	        #Retval := FC_LogMsg(EventID := 3002,
	                               EventLevel := 2,
	                               EventGroup := 33,
	                               LogMsg := DB_LogMsg.LogMsg_5);
	    END_IF;
	END_REGION
	
	//------------------------------------------------------
	// Log event when acknowledgment timeout occurs
	//------------------------------------------------------
	
	REGION Log event- acknowledgment timeout
	    IF #Communication.Log.Ack_timeout THEN
	        #Communication.Log.Ack_timeout := FALSE;
	        // Logging
	        //(LOG)3009=$ Node $, seq: $, acknowledge timeout!
	        DB_LogMsg.LogMsg_6.Para_STRING_01.Data := #Source.DecisionPoint;
	        DB_LogMsg.LogMsg_6.Para_BYTE_02.Data := #Communication.SendSeq;
	        #Retval := FC_LogMsg(EventID := 3009,
	                               EventLevel := 3,
	                               EventGroup := 33,
	                               LogMsg := DB_LogMsg.LogMsg_6);
	    END_IF;
	END_REGION
	
	
	
END_FUNCTION_BLOCK
END_NAMESPACE

NAMESPACE ProductionLine
FUNCTION_BLOCK FB_OPC_ReceiveSendAck
{ S7_Optimized_Access := 'TRUE' ; Published := 'FALSE' }
VERSION : 0.1
   VAR_IN_OUT 
      SourceSeq : Int;
      AckSeq : Int;
   END_VAR

   VAR 
      New_data_received : Bool;
      Ack_send : Bool;
      Log : Struct
         New_data_received : Bool;
         Ack_send : Bool;
      END_STRUCT;
   END_VAR


BEGIN
	// ==========================================================================================================================================
	// Company        : LogTech, s.r.o.
	// Created by     : Mahmoud Elnady
	// Block          : OPC_SendReciveAck
	// Project        : Lekarna, Chrudim -PLC001 -MCC001
	// Project number : 23-157
	// ==========================================================================================================================================
	
	// =========================
	// REGION: Acknowledgement Handling
	// =========================
	// This region handles sending an acknowledgment signal.
	// When #Ack_send is TRUE, it means an ACK needs to be sent for the last received sequence.
	// The ACK sequence is set equal to the source sequence to confirm receipt.
	// Then, #Ack_send is reset to FALSE, and a log flag is set to indicate ACK was sent.
	
	REGION Ack_Handling
	    
	    IF #Ack_send THEN
	        #AckSeq := #SourceSeq;        // Update ACK sequence to match source sequence
	        #Ack_send := FALSE;           // Reset ACK send request
	        #Log.Ack_send := TRUE;        // Set log flag for diagnostics or monitoring
	    END_IF;
	    
	END_REGION
	
	
	// =========================
	// REGION: New Data Detection
	// =========================
	// This region checks if a new data sequence has been received.
	// If the source and ACK sequences are not equal, it determines if it's truly new data:
	// - If both sequences are non-zero, or source is 1 and ACK is 0 (initial start case),
	//   then new data is considered received.
	// - Otherwise, it assumes the ACK was missed and sets ACK to current source.
	
	REGION New_Data_Detection
	    
	    IF #SourceSeq <> #AckSeq THEN
	        // Check if both sequences are valid (non-zero), or it's the initial case (1,0)
	        IF (#SourceSeq <> 0 AND #AckSeq <> 0) OR (#SourceSeq = 1 AND #AckSeq = 0) THEN
	            #New_data_received := TRUE;           // Flag new data received
	            #Log.#New_data_received := TRUE;      // Set log flag for diagnostics
	        ELSE
	            #AckSeq := #SourceSeq;                // Treat as missed ACK and sync
	        END_IF;
	    END_IF;
	    
	END_REGION
	
END_FUNCTION_BLOCK
END_NAMESPACE

NAMESPACE ProductionLine
FUNCTION_BLOCK FB_OPC_SendReciveAck
{ S7_Optimized_Access := 'TRUE' ; Published := 'FALSE' }
VERSION : 0.1
   VAR_INPUT 
      Timeout : Time;
   END_VAR

   VAR_IN_OUT 
      SourceSeq : Int;
      AckSeq : Int;
   END_VAR

   VAR 
      Send : Bool;
      New_Ack_received : Bool;
      Ack_timeout : Bool;
      Send_prev : Bool;
      SendSeq : Int;
      TimeoutTimmer {InstructionName := 'IEC_TIMER'; LibVersion := '1.0'; S7_SetPoint := 'False'} : IEC_TIMER;
      Log : Struct
         Send : Bool;
         New_Ack_received : Bool;
         Ack_timeout : Bool;
      END_STRUCT;
   END_VAR

   VAR CONSTANT 
      maxInc : Int := 9999;
   END_VAR


BEGIN
	// ==========================================================================================================================================
	// Company        : LogTech, s.r.o.
	// Created by     : Mahmoud Elnady
	// Block          : OPC_SendReciveAck
	// Project        : Lekarna, Chrudim -PLC001 -MCC001
	// Project number : 23-157
	// ==========================================================================================================================================
	
	// REGION: Handle New Send Request
	REGION Handle_Send_Request
	    // Triggered on rising edge of #Send signal
	    IF #Send AND NOT #Send_prev THEN
	         #AckSeq := 0;  // Reset acknowledgment sequence
	        
	        // Increment source sequence, wrapping around after 99999 (B#16#270F)
	         IF #SourceSeq <> #maxInc THEN
	             #SourceSeq += 1;
	         ELSE
	             #SourceSeq := 1;
	         END_IF;
	        
	        #SendSeq := #SourceSeq;       // Set current send sequence
	        #New_Ack_received := FALSE;   // Reset acknowledgment flag
	        #Log.Send := TRUE;            // Log send event
	    END_IF;
	END_REGION
	
	// REGION: Process Acknowledgment
	REGION Process_Acknowledgment
	    IF #Send THEN
	        // Check if acknowledgment is received for the current send
	        IF #AckSeq = #SendSeq THEN
	            IF #AckSeq <> 0 THEN
	                #New_Ack_received := TRUE;     // Mark new acknowledgment
	                #Ack_timeout := FALSE;         // Clear timeout flag
	                #Log.#New_Ack_received := TRUE; // Log acknowledgment
	            END_IF;
	            //#Send := FALSE;  // Reset send signal
	        END_IF;
	    END_IF;
	    
	    // Update previous send state
	    #Send_prev := #Send;
	END_REGION
	
	
	// REGION: Timeout Management and Retransmission
	REGION Handle_Send_Timeout
	    // Activate timeout timer if timeout value is set
	    IF #Timeout <> T#0s THEN
	        #TimeoutTimmer.TON(IN := #Send AND NOT #New_Ack_received ,
	                           PT := #Timeout);
	    END_IF;
	    
	    // On timeout expiration, trigger retransmission logic
	    IF #TimeoutTimmer.Q THEN
	        #Send_prev := FALSE;         // Reset previous send to retrigger
	        #Ack_timeout := TRUE;        // Mark acknowledgment timeout
	        #Log.Ack_timeout := TRUE;    // Log timeout event
	        RESET_TIMER(#TimeoutTimmer); // Reset timer
	    END_IF;
	END_REGION
	
	
	
	
END_FUNCTION_BLOCK
END_NAMESPACE

NAMESPACE ProductionLine
FUNCTION_BLOCK FB_OPC_SysStatus
{ S7_Optimized_Access := 'TRUE' ; Published := 'FALSE' }
VERSION : 0.1
   VAR_IN_OUT 
      Source : OPC_SystemStatus;
      Ack : OPC_SystStatus_Ack;
   END_VAR

   VAR 
      Comm { S7_SetPoint := 'False'} : FB_OPC_SendReciveAck;
      staSource { ExternalAccessible := 'False'; ExternalVisible := 'False'; ExternalWritable := 'False'; S7_SetPoint := 'False'} : OPC_SystemStatus;
      staAck { ExternalAccessible := 'False'; ExternalVisible := 'False'; ExternalWritable := 'False'; S7_SetPoint := 'False'} : OPC_SystStatus_Ack;
   END_VAR

   VAR_TEMP 
      Retval : Int;
   END_VAR


BEGIN
	// ==========================================================================================================================================
	// Company        : LogTech, s.r.o.
	// Created by     : Mahmoud Elnady
	// Block          : OPC_SendReciveAck
	// Project        : Lekarna, Chrudim -PLC001 -MCC001
	// Project number : 23-157
	// ==========================================================================================================================================
	
	//======================================================
	// Region: Communication Handling and Logging
	// Description: Manages the communication routine and logs
	//              events for message sending, acknowledgment
	//              reception, and acknowledgment timeout.
	//======================================================
	   
	//------------------------------------------------------
	// Call communication routine
	//------------------------------------------------------
	REGION Communication Routine
	    #Comm(SourceSeq := #staSource.SourceSeq,
	          AckSeq := #staAck.AckSeq,
	             Timeout := T#20s);
	END_REGION
	
	#Source.SourceSeq := #staSource.SourceSeq;
	#staAck.AckSeq := #Ack.AckSeq;
	
	
	//------------------------------------------------------
	// Log event when a new message is sent
	//------------------------------------------------------
	REGION Log event - new message
	    IF #Comm.Log.Send THEN
	        #Comm.Log.Send := FALSE;
	        
	        // (LOG)3001=$ Node $, new message sent, seq: $, $ $ $ $ $ $ $ $, $ $ $ $ $ $ $ $ $ $ $ $ $ $ $ $
	        DB_LogMsg.LogMsg_1.Para_BYTE_02.Data := #Source.SourceSeq;
	        
	        // Call logging function
	        #Retval := FC_LogMsg(EventID := 3007,
	                               EventLevel := 2,
	                               EventGroup := 33,
	                               LogMsg := DB_LogMsg.LogMsg_1);
	    END_IF;
	END_REGION
	
	   
	//------------------------------------------------------
	// Log event when new acknowledgment is received
	//------------------------------------------------------
	REGION  Log event-New acknowledgment
	       IF #Comm.Log.New_Ack_received THEN
	           #Comm.Log.New_Ack_received := FALSE;
	           
	           // (LOG)3008=$ Node $, acknowledge received, seq: $, WMSID: $
	           DB_LogMsg.LogMsg_2.Para_BYTE_02.Data := #Ack.AckSeq;
	           
	           // Call logging function
	           #Retval := FC_LogMsg(EventID := 3008,
	                                  EventLevel := 2,
	                                  EventGroup := 33,
	                                  LogMsg := DB_LogMsg.LogMsg_2);
	       END_IF;
	END_REGION
	
	   
	//------------------------------------------------------
	// Log event when acknowledgment timeout occurs
	//------------------------------------------------------
	REGION Log event- acknowledgment timeout
	       IF #Comm.Log.Ack_timeout THEN
	           #Comm.Log.Ack_timeout := FALSE;
	           
	           // (LOG)3009=$ Node $, seq: $, acknowledge timeout!
	           DB_LogMsg.LogMsg_3.Para_BYTE_02.Data := #Comm.SendSeq;
	           
	           // Call logging function
	           #Retval := FC_LogMsg(EventID := 3009,
	                                  EventLevel := 3,
	                                  EventGroup := 33,
	                                  LogMsg := DB_LogMsg.LogMsg_3);
	       END_IF;
	END_REGION
	    
	
	   
	   
	
END_FUNCTION_BLOCK
END_NAMESPACE

NAMESPACE ProductionLine
FUNCTION_BLOCK FB_Segments
{ S7_Optimized_Access := 'TRUE' ; Published := 'FALSE' }
VERSION : 0.1
   VAR 
      ConveyorID : Int;
      "Counter" : Int;
      FlowRackLoop1 : Array[_."B1.1.1".._."B1.23.1"] of Bool;
      FlowRackLoop2 : Array[_."B1.6.1".._."B1.18.1"] of Bool;
      Fragileloop1 : Array[_."D1.1.1".._."E1.6.1"] of Bool;
      Fragileloop2 : Array[_."D1.9.1".._."D1.10.1"] of Bool;
      cmp : Struct
         FlowRackLoop1 : Array[_."B1.1.1".._."B1.23.1"] of Bool;
         FlowRackLoop2 : Array[_."B1.6.1".._."B1.18.1"] of Bool;
         Fragileloop1 : Array[_."D1.1.1".._."E1.6.1"] of Bool;
         Fragileloop2 : Array[_."D1.9.1".._."D1.10.1"] of Bool;
      END_STRUCT;
      FlowRackLoopReadyToRun : Bool;
      FlowRackWorkPlaceLeftReadyToRun : Bool;
      FlowRackWorkPlaceRightReadyToRun : Bool;
      FragileloopReadyToRun : Bool;
   END_VAR


BEGIN
	// ==========================================================================================================================================
	// Company        : LogTech, s.r.o.
	// Created by     : Mahmoud Elnady
	// Block          : FB_Segments
	// Project        : Lekarna, Chrudim -PLC001 -MCC001
	// Project number : 23-157
	// ==========================================================================================================================================
	
	// ===============================
	// REGION: Flow rack loop
	// Purpose: Check the ReadyToRun status of conveyors and transfer units 
	//          for a flow rack section, then compare with a stored snapshot.
	// ===============================
	REGION Flow rack loop
	    
	    // ---------------------------------
	    // REGION: Conveyor Status Loop
	    // Purpose: Iterate over conveyor IDs from B1.1.1 to B1.28.1 
	    //          and store their ReadyToRun status in FlowRackLoop1 array.
	    // ---------------------------------
	   REGION Conveyor Status
	        FOR #Counter := _."B1.1.1" TO _."B1.23.1" DO
	            // Store ReadyToRun status of the current conveyor into FlowRackLoop1
	            #FlowRackLoop1[#Counter] := 
	            _.Global.DB_Global.Status.Line.ProductionLine.ReadyToRun[#Counter];
	        END_FOR;
	    END_REGION
	   
	    // ---------------------------------
	    // REGION: Transfer Unit Status Loop
	    // Purpose: Iterate over transfer unit IDs from B1.6.1 to B1.21.1 
	    //          and store their ReadyToRun status in FlowRackLoop2 array.
	    // ---------------------------------
	    REGION TransferUnit Status
	        FOR #Counter := _."B1.6.1" TO _."B1.18.1" DO
	            // Store ReadyToRun status of the current transfer unit into FlowRackLoop2
	            #FlowRackLoop2[#Counter] :=
	            _.Global.DB_Global.Status.Line.ProductionLine.ReadyToRun[#Counter];
	        END_FOR;
	    END_REGION
	    
	    // ---------------------------------
	    // REGION: Status Comparison
	    // Purpose: Check if both conveyor and transfer unit statuses 
	    //          match the previous recorded values (#cmp arrays).
	    // ---------------------------------
	    REGION Comparison
	        #FlowRackLoopReadyToRun := NOT 
	        ((#cmp.FlowRackLoop1 = #FlowRackLoop1) AND
	        (#cmp.FlowRackLoop2 = #FlowRackLoop2));
	    END_REGION
	    
	END_REGION
	
	
	// ===============================
	// REGION: Flow rack work place left
	// Purpose: ReadyToRun check for two specific conveyors on the left side.
	// ===============================
	REGION Flow rack work place left
	    #FlowRackWorkPlaceLeftReadyToRun :=
	    _.Global.DB_Global.Status.Line.ProductionLine.ReadyToRun[_."C1.4.1"] AND
	    _.Global.DB_Global.Status.Line.ProductionLine.ReadyToRun[_."C1.4.2"];
	END_REGION
	
	
	// ===============================
	// REGION: Flow rack work place right
	// Purpose: ReadyToRun check for two specific conveyors on the right side.
	// ===============================
	REGION Flow rack work place right
	    #FlowRackWorkPlaceRightReadyToRun :=
	    _.Global.DB_Global.Status.Line.ProductionLine.ReadyToRun[_."C1.2.1"] AND
	    _.Global.DB_Global.Status.Line.ProductionLine.ReadyToRun[_."C1.2.2"];
	END_REGION
	
	
	// ===============================
	// REGION: Fragile loop
	// Purpose: Same logic as Flow rack loop, but for the "fragile" product path.
	// ===============================
	REGION Fragile loop
	    
	    // ---------------------------------
	    // REGION: Conveyor Status Loop (Fragile)
	    // Purpose: Store ReadyToRun status for conveyors D1.1.1 to E1.6.1
	    // ---------------------------------
	    REGION Conveyor Status
	        FOR #Counter := _."D1.1.1" TO _."E1.6.1" DO
	            #Fragileloop1[#Counter] :=
	            _.Global.DB_Global.Status.Line.ProductionLine.ReadyToRun[#Counter];
	        END_FOR;
	    END_REGION
	    
	    // ---------------------------------
	    // REGION: Transfer Unit Status Loop (Fragile)
	    // Purpose: Store ReadyToRun status for transfer units D1.8.1 to D1.9.1
	    // ---------------------------------
	    REGION TransferUnit Status
	        FOR #Counter := _."D1.9.1" TO _."D1.10.1" DO
	            #Fragileloop2[#Counter] :=
	            _.Global.DB_Global.Status.Line.ProductionLine.ReadyToRun[#Counter];
	        END_FOR;
	    END_REGION
	    
	    // ---------------------------------
	    // REGION: Status Comparison (Fragile)
	    // Purpose: Check if current fragile loop status matches previous snapshot.
	    // ---------------------------------
	    REGION Comparison
	        #FragileloopReadyToRun := NOT
	        ((#cmp.Fragileloop1 = #Fragileloop1) AND
	        (#cmp.Fragileloop2 = #Fragileloop2));
	    END_REGION
	    
	END_REGION
	
END_FUNCTION_BLOCK
END_NAMESPACE

NAMESPACE ProductionLine
FUNCTION_BLOCK FB_Technology
{ S7_Optimized_Access := 'TRUE' ; Published := 'FALSE' }
VERSION : 0.1
   VAR 
      IP11 : String := 'IP11';
      IP12 : String := 'IP12';
      IP21 : String := 'IP21';
      IP22 : String := 'IP22';
      IP23 : String := 'IP23';
      IP31 : String := 'IP31';
      IP32 : String := 'IP32';
      IP41 : String := 'IP41';
      IP42 : String := 'IP42';
      ComDownStream : Struct
         DP1 : Bool;
         DP2 : Bool;
         DP3 : Bool;
         DP4 : Bool;
      END_STRUCT;
      ComTimmerDP1 {InstructionName := 'TON_TIME'; LibVersion := '1.0'} : TON_TIME;
      ComTimmerDP2 {InstructionName := 'TON_TIME'; LibVersion := '1.0'} : TON_TIME;
      ComTimmerDP3 {InstructionName := 'TON_TIME'; LibVersion := '1.0'} : TON_TIME;
      ComTimmerDP4 {InstructionName := 'TON_TIME'; LibVersion := '1.0'} : TON_TIME;
   END_VAR


BEGIN
	// ==========================================================================================================================================
	// Company        : LogTech, s.r.o.
	// Created by     : Mahmoud Elnady
	// Block          : FB_OPC_Communication
	// Project        : Lekarna, Chrudim -PLC001 -MCC001
	// Project number : 23-157
	// ==========================================================================================================================================
	
	REGION Destination request TO WMS
	    // Send destination request to WMS
	    REGION DP1
	        IF IDB_BarcodeReader.DP1."Dataman-Results Available" OR
	            IDB_ProductionLine."A1.5.1".CONVEYOR_SENSOR.PosEdge.Q
	        THEN
	            OPC_Data.DP1.DestRequest.Source.Barcode := IDB_BarcodeReader.DP1.ResultStr;
	            IDB_OPC_Communication.Communication_DP1.Communication.Send := TRUE;
	            #ComDownStream.DP1 := TRUE;
	        ELSIF (IDB_OPC_Communication.Communication_DP1.Communication.SourceSeq =
	            IDB_OPC_Communication.Communication_DP1.Communication.AckSeq)
	            OR #ComTimmerDP1.Q
	        THEN
	            IDB_OPC_Communication.Communication_DP1.Communication.Send := FALSE;
	        END_IF;
	         
	    END_REGION
	    
	    REGION DP2
	        IF IDB_BarcodeReader.DP2."Dataman-Results Available" OR
	            IDB_ProductionLine."B1.9.1".CONVEYOR_SENSOR.PosEdge.Q
	        THEN
	            OPC_Data.DP2.DestRequest.Source.Barcode := IDB_BarcodeReader.DP2.ResultStr;
	            IDB_OPC_Communication.Communication_DP2.Communication.Send := TRUE;
	            #ComDownStream.DP2 := TRUE;
	        ELSIF (IDB_OPC_Communication.Communication_DP2.Communication.SourceSeq =
	            IDB_OPC_Communication.Communication_DP2.Communication.AckSeq)
	            OR #ComTimmerDP2.Q
	        THEN
	            IDB_OPC_Communication.Communication_DP2.Communication.Send := FALSE;
	        END_IF;
	    END_REGION
	    
	    REGION DP3
	        IF IDB_BarcodeReader.DP3."Dataman-Results Available" OR
	            IDB_ProductionLine."B1.17.1".CONVEYOR_SENSOR.PosEdge.Q
	        THEN
	            OPC_Data.DP3.DestRequest.Source.Barcode := IDB_BarcodeReader.DP3.ResultStr;
	            IDB_OPC_Communication.Communication_DP3.Communication.Send := TRUE;
	            #ComDownStream.DP3 := TRUE;
	        ELSIF (IDB_OPC_Communication.Communication_DP3.Communication.SourceSeq =
	            IDB_OPC_Communication.Communication_DP3.Communication.AckSeq)
	            OR #ComTimmerDP3.Q
	        THEN
	            IDB_OPC_Communication.Communication_DP3.Communication.Send := FALSE;
	        END_IF;
	    END_REGION
	    
	    REGION DP4
	        IF IDB_BarcodeReader.DP4."Dataman-Results Available" OR
	            IDB_ProductionLine."A1.7.4".CONVEYOR_SENSOR.PosEdge.Q
	        THEN
	            OPC_Data.DP4.DestRequest.Source.Barcode := IDB_BarcodeReader.DP4.ResultStr;
	            IDB_OPC_Communication.Communication_DP4.Communication.Send := TRUE;
	            #ComDownStream.DP4 := TRUE;
	        ELSIF (IDB_OPC_Communication.Communication_DP4.Communication.SourceSeq =
	            IDB_OPC_Communication.Communication_DP4.Communication.AckSeq)
	            OR #ComTimmerDP4.Q
	        THEN
	            IDB_OPC_Communication.Communication_DP4.Communication.Send := FALSE;
	        END_IF;
	        
	    END_REGION
	    
	END_REGION
	
	REGION Wait FOR data from WMS
	    // Wait for data from WMS
	    REGION Mabs A1.6.1 & A1.6.2 Dir
	        IF IDB_OPC_Communication.Communication_DP1.Communication.New_Ack_received THEN
	            //IDB_OPC_Communication.Communication_DP1.Communication.New_Ack_received := FALSE;
	            #ComDownStream.DP1 := FALSE;
	            IF OPC_Data.DP1.DestRequest.Ack.Destination = #IP11 THEN
	                DB_ToteTracking.Conveyor[_."A1.5.1"].ToteDir.Straight := TRUE;
	                DB_ToteTracking.Conveyor[_."A1.5.1"].ToteDir.toRight := FALSE;
	                DB_ToteTracking.Conveyor[_."A1.2.1"].ToteDir.toLeft := FALSE;
	            ELSIF
	                OPC_Data.DP1.DestRequest.Ack.Destination = #IP12 THEN
	                DB_ToteTracking.Conveyor[_."A1.5.1"].ToteDir.toRight := TRUE;
	                DB_ToteTracking.Conveyor[_."A1.5.1"].ToteDir.Straight := FALSE;
	                DB_ToteTracking.Conveyor[_."A1.5.1"].ToteDir.toLeft := FALSE;
	            ELSE
	                DB_ToteTracking.Conveyor[_."A1.5.1"].ToteDir.Straight := FALSE;
	                DB_ToteTracking.Conveyor[_."A1.5.1"].ToteDir.toRight := FALSE;
	                DB_ToteTracking.Conveyor[_."A1.5.1"].ToteDir.toLeft := FALSE;
	            END_IF;
	        END_IF;
	    END_REGION
	    
	    REGION Transfer Unit B1.10.1 Dir
	        IF IDB_OPC_Communication.Communication_DP2.Communication.New_Ack_received THEN
	            //IDB_OPC_Communication.Communication_DP2.Communication.New_Ack_received := FALSE;
	            #ComDownStream.DP2 := FALSE;
	            IF  OPC_Data.DP2.DestRequest.Ack.Destination = #IP21 THEN
	                DB_ToteTracking.Conveyor[_."B1.9.1"].ToteDir.Straight := TRUE;
	                DB_ToteTracking.Conveyor[_."B1.9.1"].ToteDir.toRight := FALSE;
	                DB_ToteTracking.Conveyor[_."B1.9.1"].ToteDir.toLeft := FALSE;
	            ELSIF
	                (OPC_Data.DP2.DestRequest.Ack.Destination = #IP22 OR
	                OPC_Data.DP2.DestRequest.Ack.Destination = #IP23) THEN
	                DB_ToteTracking.Conveyor[_."B1.9.1"].ToteDir.toRight := TRUE;
	                DB_ToteTracking.Conveyor[_."B1.9.1"].ToteDir.Straight := FALSE;
	                DB_ToteTracking.Conveyor[_."B1.9.1"].ToteDir.toLeft := FALSE;
	                //Transfer Unit C1.1.3 Dir
	                IF OPC_Data.DP2.DestRequest.Ack.Destination = #IP22 THEN
	                    DB_ToteTracking.Transfer[_."B1.9.1"].Straight := FALSE;
	                    DB_ToteTracking.Transfer[_."B1.9.1"].toRight := TRUE;
	                    DB_ToteTracking.Transfer[_."B1.9.1"].toLeft := FALSE;
	                ELSIF  OPC_Data.DP2.DestRequest.Ack.Destination = #IP23 THEN
	                    DB_ToteTracking.Transfer[_."B1.9.1"].toRight := FALSE;
	                    DB_ToteTracking.Transfer[_."B1.9.1"].Straight := FALSE;
	                    DB_ToteTracking.Transfer[_."B1.9.1"].toLeft := TRUE;
	                ELSE
	                    DB_ToteTracking.Transfer[_."B1.9.1"].Straight := FALSE;
	                    DB_ToteTracking.Transfer[_."B1.9.1"].toRight := FALSE;
	                    DB_ToteTracking.Transfer[_."B1.9.1"].toLeft := FALSE;
	                END_IF;
	                
	            ELSE
	                DB_ToteTracking.Conveyor[_."B1.9.1"].ToteDir.Straight := FALSE;
	                DB_ToteTracking.Conveyor[_."B1.9.1"].ToteDir.toRight := FALSE;
	                DB_ToteTracking.Conveyor[_."B1.9.1"].ToteDir.toLeft := FALSE;
	            END_IF;
	        END_IF;
	    END_REGION
	    
	    
	    REGION Transfer Unit B1.21.1 Dir
	        IF IDB_OPC_Communication.Communication_DP3.Communication.New_Ack_received THEN
	            //IDB_OPC_Communication.Communication_DP3.Communication.New_Ack_received := FALSE;
	            #ComDownStream.DP3 := FALSE;
	            IF  OPC_Data.DP3.DestRequest.Ack.Destination = #IP31 THEN
	                DB_ToteTracking.Conveyor[_."B1.17.1"].ToteDir.Straight := TRUE;
	                DB_ToteTracking.Conveyor[_."B1.17.1"].ToteDir.toRight := FALSE;
	                DB_ToteTracking.Conveyor[_."B1.17.1"].ToteDir.toLeft := FALSE;
	                
	            ELSIF OPC_Data.DP3.DestRequest.Ack.Destination = #IP32 THEN
	                DB_ToteTracking.Conveyor[_."B1.17.1"].ToteDir.toRight := FALSE;
	                DB_ToteTracking.Conveyor[_."B1.17.1"].ToteDir.Straight := FALSE;
	                DB_ToteTracking.Conveyor[_."B1.17.1"].ToteDir.toLeft := TRUE;
	                
	            ELSE
	                DB_ToteTracking.Conveyor[_."B1.17.1"].ToteDir.Straight := FALSE;
	                DB_ToteTracking.Conveyor[_."B1.17.1"].ToteDir.toRight := FALSE;
	                DB_ToteTracking.Conveyor[_."B1.17.1"].ToteDir.toLeft := FALSE;
	            END_IF;
	        END_IF;
	    END_REGION
	    
	    REGION Mabs A1.8.1 & A1.8.2 Dir
	        IF IDB_OPC_Communication.Communication_DP4.Communication.New_Ack_received THEN
	            //IDB_OPC_Communication.Communication_DP4.Communication.New_Ack_received := FALSE;
	            #ComDownStream.DP4 := FALSE;
	            IF  OPC_Data.DP4.DestRequest.Ack.Destination = #IP41 THEN
	                DB_ToteTracking.Conveyor[_."A1.7.4"].ToteDir.Straight := TRUE;
	                DB_ToteTracking.Conveyor[_."A1.7.4"].ToteDir.toRight := FALSE;
	                DB_ToteTracking.Conveyor[_."A1.7.4"].ToteDir.toLeft := FALSE;
	            ELSIF
	                OPC_Data.DP4.DestRequest.Ack.Destination = #IP42 THEN
	                DB_ToteTracking.Conveyor[_."A1.7.4"].ToteDir.toRight := TRUE;
	                DB_ToteTracking.Conveyor[_."A1.7.4"].ToteDir.Straight := FALSE;
	                DB_ToteTracking.Conveyor[_."A1.7.4"].ToteDir.toLeft := FALSE;
	            ELSE
	                DB_ToteTracking.Conveyor[_."A1.7.4"].ToteDir.Straight := FALSE;
	                DB_ToteTracking.Conveyor[_."A1.7.4"].ToteDir.toRight := FALSE;
	                DB_ToteTracking.Conveyor[_."A1.7.4"].ToteDir.toLeft := FALSE;
	            END_IF;
	        END_IF;
	    END_REGION
	    
	    REGION Wait WMS Response
	        #ComTimmerDP1(IN := #ComDownStream.DP1,
	                      PT := t#45s);
	        
	        IF #ComTimmerDP1.Q THEN
	            #ComDownStream.DP1 := FALSE;
	        END_IF;
	        
	        #ComTimmerDP2(IN := #ComDownStream.DP2,
	                      PT := t#45s);
	        
	        IF #ComTimmerDP2.Q THEN
	            #ComDownStream.DP2 := FALSE;
	        END_IF;
	        
	        #ComTimmerDP3(IN := #ComDownStream.DP3,
	                      PT := t#45s);
	        
	        IF #ComTimmerDP3.Q THEN
	            #ComDownStream.DP3 := FALSE;
	        END_IF;
	        
	        #ComTimmerDP4(IN := #ComDownStream.DP4,
	                      PT := t#45s);
	        
	        IF #ComTimmerDP4.Q THEN
	            #ComDownStream.DP4 := FALSE;
	        END_IF;
	        
	    END_REGION
	
	END_REGION
	
	
	REGION Destination info TO WMS
	    // Send destination info to WMS
	    REGION IP1
	        IF IDB_ProductionLine."A1.7.2".CONVEYOR_SENSOR.PosEdge.Q AND
	            NOT IDB_OPC_Communication.Communication_IP1.Communication.Send THEN
	            OPC_Data.IP1.DestInfo.Source.Barcode := DB_ToteTracking.Conveyor[_."A1.7.1"].Barcode;
	            OPC_Data.IP1.DestInfo.Source.InformationPoint := #IP11;
	            IDB_OPC_Communication.Communication_IP1.Communication.Send := TRUE;
	        END_IF;
	        
	    END_REGION
	    REGION IP2
	        IF IDB_ProductionLine."B1.2.1".CONVEYOR_SENSOR.PosEdge.Q AND
	            NOT IDB_OPC_Communication.Communication_IP2.Communication.Send THEN
	            OPC_Data.IP2.DestInfo.Source.Barcode := DB_ToteTracking.Conveyor[_."B1.1.1"].Barcode;
	            OPC_Data.IP2.DestInfo.Source.InformationPoint := #IP12;
	            IDB_OPC_Communication.Communication_IP2.Communication.Send := TRUE;
	        END_IF;
	        
	    END_REGION
	    
	    REGION IP3
	        IF IDB_ProductionLine."B1.11.2".CONVEYOR_SENSOR.PosEdge.Q AND
	            NOT IDB_OPC_Communication.Communication_IP3.Communication.Send THEN
	            OPC_Data.IP3.DestInfo.Source.Barcode := DB_ToteTracking.Conveyor[_."B1.11.1"].Barcode;
	            OPC_Data.IP3.DestInfo.Source.InformationPoint := #IP21;
	            IDB_OPC_Communication.Communication_IP3.Communication.Send := TRUE;
	        END_IF;
	    END_REGION
	    
	    REGION IP4
	        IF IDB_ProductionLine."C1.2.1".CONVEYOR_SENSOR.PosEdge.Q AND
	            NOT IDB_OPC_Communication.Communication_IP4.Communication.Send THEN
	            OPC_Data.IP4.DestInfo.Source.Barcode := DB_ToteTracking.Conveyor[_."C1.2.2"].Barcode;
	            OPC_Data.IP4.DestInfo.Source.InformationPoint := #IP22;
	            IDB_OPC_Communication.Communication_IP4.Communication.Send := TRUE;
	        END_IF;
	        
	    END_REGION
	    
	    REGION IP5
	        IF IDB_ProductionLine."C1.4.2".CONVEYOR_SENSOR.PosEdge.Q AND
	            NOT IDB_OPC_Communication.Communication_IP5.Communication.Send THEN
	            OPC_Data.IP5.DestInfo.Source.Barcode := DB_ToteTracking.Conveyor[_."C1.4.1"].Barcode;
	            OPC_Data.IP5.DestInfo.Source.InformationPoint := #IP23;
	            IDB_OPC_Communication.Communication_IP5.Communication.Send := TRUE;
	        END_IF;
	        
	    END_REGION
	    
	    REGION IP6
	        IF IDB_ProductionLine."B1.20.1".CONVEYOR_SENSOR.PosEdge.Q AND
	            NOT IDB_OPC_Communication.Communication_IP6.Communication.Send THEN
	            OPC_Data.IP6.DestInfo.Source.Barcode := DB_ToteTracking.Conveyor[_."B1.19.1"].Barcode;
	            OPC_Data.IP6.DestInfo.Source.InformationPoint := #IP31;
	            IDB_OPC_Communication.Communication_IP6.Communication.Send := TRUE;
	        END_IF;
	    END_REGION
	    
	    REGION IP7
	        IF (IDB_ProductionLine."B1.6.1"."Left/RightSensor" OR 
	            _.ProductionLine.IDB_Flow_Test.R_TRIG_Instance.Q) AND //only for simulation purpose 
	            NOT IDB_OPC_Communication.Communication_IP7.Communication.Send THEN
	            OPC_Data.IP7.DestInfo.Source.Barcode := DB_ToteTracking.Conveyor[_."B1.6.1"].Barcode;
	            OPC_Data.IP7.DestInfo.Source.InformationPoint := #IP32;
	            IDB_OPC_Communication.Communication_IP7.Communication.Send := TRUE;
	        END_IF;
	        
	    END_REGION
	    
	    REGION IP8
	        IF IDB_ProductionLine."A1.10.2".CONVEYOR_SENSOR.PosEdge.Q AND
	            NOT IDB_OPC_Communication.Communication_IP8.Communication.Send THEN
	            OPC_Data.IP8.DestInfo.Source.Barcode := DB_ToteTracking.Conveyor[_."A1.10.1"].Barcode;
	            OPC_Data.IP8.DestInfo.Source.InformationPoint := #IP41;
	            IDB_OPC_Communication.Communication_IP8.Communication.Send := TRUE;
	        END_IF;
	    END_REGION
	    
	    REGION IP9
	        IF IDB_ProductionLine."D1.2.1".CONVEYOR_SENSOR.PosEdge.Q AND
	            NOT IDB_OPC_Communication.Communication_IP9.Communication.Send THEN
	            OPC_Data.IP9.DestInfo.Source.Barcode := DB_ToteTracking.Conveyor[_."D1.1.1"].Barcode;
	            OPC_Data.IP9.DestInfo.Source.InformationPoint := #IP42;
	            IDB_OPC_Communication.Communication_IP9.Communication.Send := TRUE;
	        END_IF;
	    END_REGION
	    
	    
	END_REGION
	
	
	REGION Wait FOR data from WMS
	    // Wait for data from WMS
	    REGION IP1 Ack
	        IF IDB_OPC_Communication.Communication_IP1.Communication.New_Ack_received THEN
	            IDB_OPC_Communication.Communication_IP1.Communication.Send := FALSE;
	            IDB_OPC_Communication.Communication_IP1.Communication.New_Ack_received := FALSE;
	        END_IF;
	    END_REGION
	    
	    REGION IP2 Ack
	        IF IDB_OPC_Communication.Communication_IP2.Communication.New_Ack_received THEN
	            IDB_OPC_Communication.Communication_IP2.Communication.Send := FALSE;
	            IDB_OPC_Communication.Communication_IP2.Communication.New_Ack_received := FALSE;
	        END_IF;
	    END_REGION
	    
	    REGION IP3 Ack
	        IF IDB_OPC_Communication.Communication_IP3.Communication.New_Ack_received THEN
	            IDB_OPC_Communication.Communication_IP3.Communication.Send := FALSE;
	            IDB_OPC_Communication.Communication_IP3.Communication.New_Ack_received := FALSE;
	        END_IF;
	    END_REGION
	    
	    REGION IP4 Ack
	        IF IDB_OPC_Communication.Communication_IP4.Communication.New_Ack_received THEN
	            IDB_OPC_Communication.Communication_IP4.Communication.Send := FALSE;
	            IDB_OPC_Communication.Communication_IP4.Communication.New_Ack_received := FALSE;
	        END_IF;
	    END_REGION
	    
	    REGION IP5 Ack
	        IF IDB_OPC_Communication.Communication_IP5.Communication.New_Ack_received THEN
	            IDB_OPC_Communication.Communication_IP5.Communication.Send := FALSE;
	            IDB_OPC_Communication.Communication_IP5.Communication.New_Ack_received := FALSE;
	        END_IF;
	    END_REGION
	    
	    REGION IP6 Ack
	        IF IDB_OPC_Communication.Communication_IP6.Communication.New_Ack_received THEN
	            IDB_OPC_Communication.Communication_IP6.Communication.Send := FALSE;
	            IDB_OPC_Communication.Communication_IP6.Communication.New_Ack_received := FALSE;
	        END_IF;
	    END_REGION
	    
	    REGION IP7 Ack
	        IF IDB_OPC_Communication.Communication_IP7.Communication.New_Ack_received THEN
	            IDB_OPC_Communication.Communication_IP7.Communication.Send := FALSE;
	            IDB_OPC_Communication.Communication_IP7.Communication.New_Ack_received := FALSE;
	        END_IF;
	    END_REGION
	    
	    REGION IP8 Ack
	        IF IDB_OPC_Communication.Communication_IP8.Communication.New_Ack_received THEN
	            IDB_OPC_Communication.Communication_IP8.Communication.Send := FALSE;
	            IDB_OPC_Communication.Communication_IP8.Communication.New_Ack_received := FALSE;
	        END_IF;
	    END_REGION
	    
	    REGION IP9 Ack
	        IF IDB_OPC_Communication.Communication_IP9.Communication.New_Ack_received THEN
	            IDB_OPC_Communication.Communication_IP9.Communication.Send := FALSE;
	            IDB_OPC_Communication.Communication_IP9.Communication.New_Ack_received := FALSE;
	        END_IF;
	    END_REGION
	    
	END_REGION
	
	
	
	
	
	
	
	
	
	   
	        
	         
END_FUNCTION_BLOCK
END_NAMESPACE

NAMESPACE ProductionLine
FUNCTION FC_LogMsg : Int
{ S7_Optimized_Access := 'TRUE' ; Published := 'FALSE' }
VERSION : 0.1
   VAR_INPUT 
      EventID : Int;
      EventLevel : Byte;
      EventGroup : Byte;
      LogMsg : Variant;
   END_VAR

   VAR_TEMP 
      LtLogMsg : Log_LogMsg_Header;
      LabyAuxBuffer : Array[0..1023] of Byte;
      LdiMsgPosition : DInt;
      LdiMsgStartPosition : DInt;
      LiReturn : Int;
   END_VAR

   VAR CONSTANT 
      coSTX : Byte := 16#2;
      coSOH : Byte := 16#1;
      coMsgType_Log : Byte := 16#5;
      LOGMSG_BUFFER_SIZE : Int := 8191;
   END_VAR


BEGIN
	// ==========================================================================================================================================
	// Company        : LogTech, s.r.o.
	// Created by     : Mahmoud Elnady
	// Block          : OPC_SendReciveAck
	// Project        : Lekarna, Chrudim -PLC001 -MCC001
	// Project number : 23-157
	// ==========================================================================================================================================
	
	
	#LtLogMsg.STX := #coSTX;                              // initialisation of fixed header fields
	#LtLogMsg.SOH := #coSOH;
	#LtLogMsg.MsgType := #coMsgType_Log;
	
	#LtLogMsg.EventLevel := #EventLevel;                 // write input parameters into message header
	#LtLogMsg.EventGroup := #EventGroup;
	#LtLogMsg.EventID := #EventID;
	
	#LtLogMsg.MsgLength := 0;                               // initialisation of message length in header
	#LdiMsgPosition := 0;                                   // initialisation of write position in auxiliary buffer
	
	// !!! how to get timestamp with less cycle time consumption ???
	#LiReturn := RD_LOC_T(#LtLogMsg.Timestamp);            // write system date and time into message header
	
	// write message header into auxiliary buffer (message length in header still invalid!)
	#FC_LogMsg := Serialize(SRC_VARIABLE := #LtLogMsg, DEST_ARRAY => #LabyAuxBuffer, POS := #LdiMsgPosition);
	IF #FC_LogMsg <> 0 THEN
	    RETURN;                 // instruction faulted - error status returned in iRetVal
	END_IF;
	
	// write message data into auxiliary buffer
	#FC_LogMsg := Serialize(SRC_VARIABLE := #LogMsg, DEST_ARRAY => #LabyAuxBuffer, POS := #LdiMsgPosition);
	IF #FC_LogMsg <> 0 THEN
	    RETURN;                 // instruction faulted - error status returned in iRetVal
	END_IF;
	
	// check if the message data fits in the buffer
	IF DB_LogMsg.Write_Position + DINT_TO_INT(#LdiMsgPosition) > #LOGMSG_BUFFER_SIZE THEN
	    RETURN;
	END_IF;
	
	#LtLogMsg.MsgLength := DINT_TO_INT(#LdiMsgPosition);    // write message length into message header
	
	#LabyAuxBuffer[2] := #LtLogMsg.MsgLength.%B0;            // and write it bytewise into appropriate position in auxiliary buffer
	#LabyAuxBuffer[3] := #LtLogMsg.MsgLength.%B1;
	
	// ^^^ REPLACED with previous lines ^^^
	// overwrite the message header in buffer with valid message length
	// #LogMsg := Serialize(SRC_VARIABLE := #tHeader, DEST_ARRAY => "LogMsg_DB".abyLogMsg_Buffer, POS := #LdiMsgStartPosition);
	// IF #LogMsg <> 0 THEN
	//     RETURN;                 // instruction faulted - error status returned in iRetVal
	// END_IF;
	
	// ! INTERRUPT DISABLED !
	#LiReturn := DIS_IRT(MODE := 0, OB_NR := 0);
	
	MOVE_BLK(IN := #LabyAuxBuffer[0],
	         COUNT := DINT_TO_ULINT(#LdiMsgPosition),
	         OUT => DB_LogMsg.abyLogMsg_Buffer[DB_LogMsg.Write_Position]);
	
	DB_LogMsg.Write_Position := DB_LogMsg.Write_Position + DINT_TO_INT(#LdiMsgPosition);    // if everything was ok, update the write position in buffer
	
	// ! INTERRUPT ENABLE !
	#LiReturn := EN_IRT(MODE := 0, OB_NR := 0);
	
	// !!! all messages since last send are in "LogMsg_DB".abyLogMsg_Buffer - somewhere must be function to send these data to log server
	// !!! is this safe for interrupt(s) ? and optimal ?
	// !!! what about sequence number ? should we have one ?
	// !!! solution for buffer overflow !
	
END_FUNCTION
END_NAMESPACE

NAMESPACE ProductionLine
FUNCTION_BLOCK FB_ToteTracking
{ S7_Optimized_Access := 'TRUE' ; Published := 'FALSE' }
VERSION : 0.1
   VAR 
      ZoneBpJam_Occ {InstructionName := 'TON_TIME'; LibVersion := '1.0'; S7_SetPoint := 'False'} : TON_TIME;
      ZoneBpJam_NotOcc {InstructionName := 'TON_TIME'; LibVersion := '1.0'} : TON_TIME;
      DivertToManual { S7_SetPoint := 'True'} : Bool;
      HoldDivertToManual : Bool;
      "RT_Exit_1_" {InstructionName := 'R_TRIG'; LibVersion := '1.0'; S7_SetPoint := 'False'} : Array[1..1] of R_TRIG;
      "RT_Exit_2_" {InstructionName := 'R_TRIG'; LibVersion := '1.0'; S7_SetPoint := 'False'} : Array[1..6] of R_TRIG;
      NoReadTote { S7_SetPoint := 'True'} : String := 'BOX-9999-99999';
      NoData : Array[1..6] of Bool;
   END_VAR


BEGIN
	// ==========================================================================================================================================
	// Company        : LogTech, s.r.o.
	// Created by     : Anton Vinoth Soundraraj
	// Block          : FB_CreatePostData
	// Project        : Gurkerl, Vienna -PLC001 -MCC100
	// Project number : 23-158
	// ==========================================================================================================================================
	
	REGION A1.5.1
	    
	    // write barcode data
	    DB_ToteTracking.Conveyor[_."A1.5.1"].Barcode :=
	    IDB_BarcodeReader.DP1.ResultStr;
	    
	END_REGION
	
	
	REGION A1.5.2
	    
	    IF IDB_ProductionLine."A1.5.1".CONVEYOR_SENSOR.SensorEdge.Negative THEN
	        // Barcode
	        DB_ToteTracking.Conveyor[_."A1.5.2"].Barcode :=
	        DB_ToteTracking.Conveyor[_."A1.5.1"].Barcode;
	        // main diverter direction
	        DB_ToteTracking.Conveyor[_."A1.5.2"].ToteDir :=
	        DB_ToteTracking.Conveyor[_."A1.5.1"].ToteDir;
	    END_IF;
	    
	END_REGION
	
	
	REGION A1.5.3
	    
	    IF IDB_ProductionLine."A1.5.2".CONVEYOR_SENSOR.SensorEdge.Negative
	    THEN
	        // Barcode
	        DB_ToteTracking.Conveyor[_."A1.5.3"].Barcode :=
	        DB_ToteTracking.Conveyor[_."A1.5.2"].Barcode;
	        // main diverter direction
	        DB_ToteTracking.Conveyor[_."A1.5.3"].ToteDir :=
	        DB_ToteTracking.Conveyor[_."A1.5.2"].ToteDir;
	    END_IF;
	    
	    
	    REGION Decision: main diverter: before Mabs
	        
	        // to Right
	        IF DB_ToteTracking.Conveyor[_."A1.5.3"].ToteDir.toRight OR
	            (DB_ToteTracking.Conveyor[_."A1.5.3"].Barcode = #NoReadTote) OR // bad read tote
	            _.Global.IDB_HardwareDiag."Cognex -10.106.129.24".CommunicationError // Cognex reader communcation error
	        THEN
	            DB_ToteTracking.Conveyor[_."A1.6.1"].ToteDir.Straight := FALSE;
	            DB_ToteTracking.Conveyor[_."A1.6.1"].ToteDir.toRight := TRUE;
	            DB_ToteTracking.Conveyor[_."A1.6.2"].ToteDir.Straight := FALSE;
	            DB_ToteTracking.Conveyor[_."A1.6.2"].ToteDir.toRight := TRUE;
	        END_IF;
	        // to straight
	        IF DB_ToteTracking.Conveyor[_."A1.5.3"].ToteDir.Straight AND
	            NOT (DB_ToteTracking.Conveyor[_."A1.5.3"].Barcode = #NoReadTote) AND // good read tote
	            NOT _.Global.IDB_HardwareDiag."Cognex -10.106.129.24".CommunicationError // Keyence reader communcation error
	        THEN
	            DB_ToteTracking.Conveyor[_."A1.6.1"].ToteDir.Straight := TRUE;
	            DB_ToteTracking.Conveyor[_."A1.6.1"].ToteDir.toRight := FALSE;
	            DB_ToteTracking.Conveyor[_."A1.6.2"].ToteDir.Straight := TRUE;
	            DB_ToteTracking.Conveyor[_."A1.6.2"].ToteDir.toRight := FALSE;
	        END_IF;
	        
	    END_REGION
	    
	END_REGION
	
	REGION B1.1.1 Right
	    
	    IF  //IDB_ProductionLine."A1.6.1".CROSS_SENSOR_FILTER.SensorEdge.Negative AND
	        IDB_ProductionLine."A1.6.1".CROSS_SENSOR_FILTER.NegEdge.Q AND
	        NOT IDB_ProductionLine."A1.6.1".CurrentPosition.right AND // remove not
	        NOT IDB_ProductionLine."A1.6.2".CurrentPosition.right //AND // remove not
	        //NOT IDB_ProductionLine."B1.1.1".ReadConveyorStatus.Occupied 
	    THEN
	        // Barcode
	        DB_ToteTracking.Conveyor[_."B1.1.1"].Barcode :=
	        DB_ToteTracking.Conveyor[_."A1.5.3"].Barcode;
	    END_IF;
	    
	END_REGION
	
	REGION B1.2.1
	    
	    IF  IDB_ProductionLine."B1.1.1".CONVEYOR_SENSOR.SensorEdge.Negative THEN
	        DB_ToteTracking.Conveyor[_."B1.2.1"] :=DB_ToteTracking.Conveyor[_."B1.1.1"];
	    END_IF;
	    
	END_REGION
	
	REGION B1.3.1
	    
	    IF IDB_ProductionLine."B1.2.1".CONVEYOR_SENSOR.SensorEdge.Negative THEN
	        DB_ToteTracking.Conveyor[_."B1.3.1"] := DB_ToteTracking.Conveyor[_."B1.2.1"];
	    END_IF;
	    
	END_REGION
	
	
	REGION A1.7.1 Straight
	    
	    IF  IDB_ProductionLine."A1.6.1".CROSS_SENSOR_FILTER.SensorEdge.Negative AND
	        NOT IDB_ProductionLine."A1.6.1".CurrentPosition.straight AND  //remove Not
	        NOT IDB_ProductionLine."A1.6.2".CurrentPosition.straight //AND  // remove Not
	        //NOT IDB_ProductionLine."A1.7.1".ReadConveyorStatus.Occupied
	    THEN
	        // Barcode
	        DB_ToteTracking.Conveyor[_."A1.7.1"].Barcode :=
	        DB_ToteTracking.Conveyor[_."A1.5.3"].Barcode;
	    END_IF;
	    
	END_REGION
	
	REGION A1.7.2
	    
	    IF IDB_ProductionLine."A1.7.1".CONVEYOR_SENSOR.SensorEdge.Negative THEN
	        DB_ToteTracking.Conveyor[_."A1.7.2"] := DB_ToteTracking.Conveyor[_."A1.7.1"];
	    END_IF;
	    
	END_REGION
	
	REGION A1.7.3
	    
	    IF IDB_ProductionLine."A1.7.2".CONVEYOR_SENSOR.SensorEdge.Negative THEN
	        DB_ToteTracking.Conveyor[_."A1.7.3"] := DB_ToteTracking.Conveyor[_."A1.7.2"];
	    END_IF;
	    
	END_REGION
	
	/////////////////////////////////////////////////////////
	//DP2
	////////////////////////////////////////////////////////
	
	REGION B1.9.1
	    
	    // write barcode data
	    DB_ToteTracking.Conveyor[_."B1.9.1"].Barcode :=
	    IDB_BarcodeReader.DP2.ResultStr;
	    
	END_REGION
	
	REGION B1.9.2
	    
	    IF IDB_ProductionLine."B1.9.1".CONVEYOR_SENSOR.SensorEdge.Negative
	    THEN
	        // Barcode
	        DB_ToteTracking.Conveyor[_."B1.9.2"].Barcode :=
	        DB_ToteTracking.Conveyor[_."B1.9.1"].Barcode;
	        // main diverter direction
	        DB_ToteTracking.Conveyor[_."B1.9.2"].ToteDir :=
	        DB_ToteTracking.Conveyor[_."B1.9.1"].ToteDir;
	        //
	        DB_ToteTracking.Transfer[_."B1.9.2"] :=
	        DB_ToteTracking.Transfer[_."B1.9.1"];
	    END_IF;
	    
	    
	    REGION Decision: second diverter: before Transfer Unit 
	        
	        // to Right for Transfer Unit B1.10.1
	        IF DB_ToteTracking.Conveyor[_."B1.9.2"].ToteDir.toRight OR
	           (DB_ToteTracking.Conveyor[_."B1.9.2"].Barcode = #NoReadTote) OR // Good read tote
	           _.Global.IDB_HardwareDiag."Cognex -10.106.129.24".CommunicationError // Cognex reader communcation error
	        THEN
	            DB_ToteTracking.Conveyor[_."B1.10.1"].ToteDir.Straight := FALSE;
	            DB_ToteTracking.Conveyor[_."B1.10.1"].ToteDir.toRight := TRUE;
	        END_IF;
	        // to straight for Transfer Unit B1.10.1 
	        IF DB_ToteTracking.Conveyor[_."B1.9.2"].ToteDir.Straight AND
	           NOT (DB_ToteTracking.Conveyor[_."B1.9.2"].Barcode = #NoReadTote) AND // Bad read tote
	           NOT _.Global.IDB_HardwareDiag."Cognex -10.106.129.24".CommunicationError // Cognex reader communcation error
	        THEN
	            DB_ToteTracking.Conveyor[_."B1.10.1"].ToteDir.Straight := TRUE;
	            DB_ToteTracking.Conveyor[_."B1.10.1"].ToteDir.toRight := FALSE;
	        END_IF;
	        
	        // to Right for Transfer Unit C1.1.3
	        IF DB_ToteTracking.Transfer[_."B1.9.2"].toRight THEN
	            DB_ToteTracking.Conveyor[_."C1.3.1"].ToteDir.toLeft := FALSE;
	            DB_ToteTracking.Conveyor[_."C1.3.1"].ToteDir.toRight := TRUE;
	        END_IF;
	        // to Left for Transfer Unit C1.1.3
	        IF DB_ToteTracking.Transfer[_."B1.9.2"].toLeft THEN
	            DB_ToteTracking.Conveyor[_."C1.3.1"].ToteDir.toLeft := TRUE;
	            DB_ToteTracking.Conveyor[_."C1.3.1"].ToteDir.toRight := FALSE;
	        END_IF;
	        
	    END_REGION
	    
	END_REGION
	
	REGION C1.1.3 Right
	    
	    IF IDB_ProductionLine."B1.10.1".FilteredSensor AND
	        DB_ToteTracking.Conveyor[_."B1.10.1"].ToteDir.toRight AND
	        NOT IDB_ProductionLine."C1.3.1".ReadTransferStatus.Occupied
	    THEN
	        // Barcode
	        DB_ToteTracking.Conveyor[_."C1.3.1"].Barcode :=
	        DB_ToteTracking.Conveyor[_."B1.9.2"].Barcode;
	    END_IF;
	    
	END_REGION
	
	REGION B1.11.1 Straight
	    
	    IF IDB_ProductionLine."B1.10.1".FilteredSensor AND
	        DB_ToteTracking.Conveyor[_."B1.10.1"].ToteDir.Straight AND
	        NOT IDB_ProductionLine."B1.11.1".ReadConveyorStatus.Occupied
	    THEN
	        // Barcode
	        DB_ToteTracking.Conveyor[_."B1.11.1"].Barcode :=
	        DB_ToteTracking.Conveyor[_."B1.9.2"].Barcode;
	    END_IF;
	    
	END_REGION
	
	REGION C1.2.2
	    IF IDB_ProductionLine."C1.3.1".FilteredSensor AND
	        DB_ToteTracking.Conveyor[_."C1.3.1"].ToteDir.toRight AND
	        NOT IDB_ProductionLine."C1.2.2".ReadConveyorStatus.Occupied
	    THEN
	        DB_ToteTracking.Conveyor[_."C1.2.2"].Barcode :=
	        DB_ToteTracking.Conveyor[_."C1.3.1"].Barcode;
	    END_IF;
	    
	END_REGION
	
	REGION C1.4.1
	    IF IDB_ProductionLine."C1.3.1".FilteredSensor AND
	        DB_ToteTracking.Conveyor[_."C1.3.1"].ToteDir.toLeft  //AND
	        //NOT IDB_ProductionLine."C1.4.1".ReadConveyorStatus.Occupied
	    THEN
	        DB_ToteTracking.Conveyor[_."C1.4.1"].Barcode :=
	        DB_ToteTracking.Conveyor[_."C1.3.1"].Barcode;
	    END_IF;
	    
	END_REGION
	
	
	/////////////////////////////////////////////////////////
	//DP3
	////////////////////////////////////////////////////////
	
	REGION B1.17.1
	    
	    // write barcode data
	    DB_ToteTracking.Conveyor[_."B1.17.1"].Barcode :=
	    IDB_BarcodeReader.DP3.ResultStr;
	    
	END_REGION
	
	REGION B1.17.2
	    
	    IF IDB_ProductionLine."B1.17.1".CONVEYOR_SENSOR.SensorEdge.Negative THEN
	        // Barcode
	        DB_ToteTracking.Conveyor[_."B1.17.2"].Barcode :=
	        DB_ToteTracking.Conveyor[_."B1.17.1"].Barcode;
	        // main diverter direction
	        DB_ToteTracking.Conveyor[_."B1.17.2"].ToteDir :=
	        DB_ToteTracking.Conveyor[_."B1.17.1"].ToteDir;
	    END_IF;
	    
	END_REGION
	
	REGION B1.17.3
	    
	    IF IDB_ProductionLine."B1.17.2".CONVEYOR_SENSOR.SensorEdge.Negative THEN
	        // Barcode
	        DB_ToteTracking.Conveyor[_."B1.17.3"].Barcode :=
	        DB_ToteTracking.Conveyor[_."B1.17.2"].Barcode;
	        // main diverter direction
	        DB_ToteTracking.Conveyor[_."B1.17.3"].ToteDir :=
	        DB_ToteTracking.Conveyor[_."B1.17.2"].ToteDir;
	    END_IF;
	    
	END_REGION
	
	
	REGION B1.17.4
	    
	    IF IDB_ProductionLine."B1.17.3".CONVEYOR_SENSOR.SensorEdge.Negative
	    THEN
	        // Barcode
	        DB_ToteTracking.Conveyor[_."B1.17.4"].Barcode :=
	        DB_ToteTracking.Conveyor[_."B1.17.3"].Barcode;
	        // main diverter direction
	        DB_ToteTracking.Conveyor[_."B1.17.4"].ToteDir :=
	        DB_ToteTracking.Conveyor[_."B1.17.3"].ToteDir;
	    END_IF;
	    
	    
	    REGION Decision: Third diverter: before Transfer Unit 
	        
	        // to Left
	        IF DB_ToteTracking.Conveyor[_."B1.17.4"].ToteDir.toLeft OR
	           (DB_ToteTracking.Conveyor[_."B1.17.4"].Barcode = #NoReadTote) OR // bad read tote
	            _.Global.IDB_HardwareDiag."Cognex -10.106.129.24".CommunicationError // Cognex reader communcation error
	        THEN
	            DB_ToteTracking.Conveyor[_."B1.18.1"].ToteDir.Straight := FALSE;
	            DB_ToteTracking.Conveyor[_."B1.18.1"].ToteDir.toLeft := TRUE;
	        END_IF;
	        // to straight
	        IF DB_ToteTracking.Conveyor[_."B1.17.4"].ToteDir.Straight AND
	            NOT (DB_ToteTracking.Conveyor[_."B1.17.4"].Barcode = #NoReadTote) AND // Good read tote
	            NOT _.Global.IDB_HardwareDiag."Cognex -10.106.129.24".CommunicationError // Cognex reader communcation error
	        THEN
	            DB_ToteTracking.Conveyor[_."B1.18.1"].ToteDir.Straight := TRUE;
	            DB_ToteTracking.Conveyor[_."B1.18.1"].ToteDir.toLeft := FALSE;
	        END_IF;
	        
	    END_REGION
	    
	END_REGION
	
	REGION B1.6.1 Left
	    
	    IF IDB_ProductionLine."B1.18.1".FilteredSensor AND
	        DB_ToteTracking.Conveyor[_."B1.18.1"].ToteDir.toLeft AND
	        NOT IDB_ProductionLine."B1.6.1".ReadTransferStatus.Occupied
	    THEN
	        // Barcode
	        DB_ToteTracking.Conveyor[_."B1.6.1"].Barcode :=
	        DB_ToteTracking.Conveyor[_."B1.17.4"].Barcode;
	    END_IF;
	    
	END_REGION
	
	REGION B1.19.1 Straight
	    
	    IF IDB_ProductionLine."B1.18.1".FilteredSensor AND
	        DB_ToteTracking.Conveyor[_."B1.18.1"].ToteDir.Straight AND
	        NOT IDB_ProductionLine."B1.19.1".ReadConveyorStatus.Occupied
	    THEN
	        // Barcode
	        DB_ToteTracking.Conveyor[_."B1.19.1"].Barcode :=
	        DB_ToteTracking.Conveyor[_."B1.17.4"].Barcode;
	    END_IF;
	    
	END_REGION
	
	/////////////////////////////////////////////////////////
	//DP4
	////////////////////////////////////////////////////////
	
	REGION A1.7.4
	    
	    // write barcode data
	    DB_ToteTracking.Conveyor[_."A1.7.4"].Barcode :=
	    IDB_BarcodeReader.DP4.ResultStr;
	    
	END_REGION
	
	REGION A1.7.5
	    
	    IF IDB_ProductionLine."A1.7.4".CONVEYOR_SENSOR.SensorEdge.Negative THEN
	        // Barcode
	        DB_ToteTracking.Conveyor[_."A1.7.5"].Barcode :=
	        DB_ToteTracking.Conveyor[_."A1.7.4"].Barcode;
	        // main diverter direction
	        DB_ToteTracking.Conveyor[_."A1.7.5"].ToteDir :=
	        DB_ToteTracking.Conveyor[_."A1.7.4"].ToteDir;
	    END_IF;
	    
	END_REGION
	
	REGION A1.7.6
	    
	    IF IDB_ProductionLine."A1.7.5".CONVEYOR_SENSOR.SensorEdge.Negative THEN
	        // Barcode
	        DB_ToteTracking.Conveyor[_."A1.7.6"].Barcode :=
	        DB_ToteTracking.Conveyor[_."A1.7.5"].Barcode;
	        // main diverter direction
	        DB_ToteTracking.Conveyor[_."A1.7.6"].ToteDir :=
	        DB_ToteTracking.Conveyor[_."A1.7.5"].ToteDir;
	    END_IF;
	    
	END_REGION
	
	
	REGION A1.8.1
	    
	    IF IDB_ProductionLine."A1.7.6".CONVEYOR_SENSOR.SensorEdge.Negative
	    THEN
	        // Barcode
	        DB_ToteTracking.Conveyor[_."A1.8.1"].Barcode :=
	        DB_ToteTracking.Conveyor[_."A1.7.6"].Barcode;
	        // main diverter direction
	        DB_ToteTracking.Conveyor[_."A1.8.1"].ToteDir :=
	        DB_ToteTracking.Conveyor[_."A1.7.6"].ToteDir;
	    END_IF;
	    
	    
	    REGION Decision: main diverter: before Mabs
	        
	        // to Right
	        IF DB_ToteTracking.Conveyor[_."A1.8.1"].ToteDir.toRight OR
	            (DB_ToteTracking.Conveyor[_."A1.8.1"].Barcode = #NoReadTote) OR // bad read tote
	            _.Global.IDB_HardwareDiag."Cognex -10.106.129.24".CommunicationError // Cognex reader communcation error
	        THEN
	            DB_ToteTracking.Conveyor[_."A1.9.1"].ToteDir.Straight := FALSE;
	            DB_ToteTracking.Conveyor[_."A1.9.1"].ToteDir.toRight := TRUE;
	            DB_ToteTracking.Conveyor[_."A1.9.2"].ToteDir.Straight := FALSE;
	            DB_ToteTracking.Conveyor[_."A1.9.2"].ToteDir.toRight := TRUE;
	        END_IF;
	        // to straight
	        IF DB_ToteTracking.Conveyor[_."A1.8.1"].ToteDir.Straight AND
	            NOT (DB_ToteTracking.Conveyor[_."A1.8.1"].Barcode = #NoReadTote) AND // good read tote
	            NOT _.Global.IDB_HardwareDiag."Cognex -10.106.129.24".CommunicationError // Keyence reader communcation error
	        THEN
	            DB_ToteTracking.Conveyor[_."A1.9.1"].ToteDir.Straight := TRUE;
	            DB_ToteTracking.Conveyor[_."A1.9.1"].ToteDir.toRight := FALSE;
	            DB_ToteTracking.Conveyor[_."A1.9.2"].ToteDir.Straight := TRUE;
	            DB_ToteTracking.Conveyor[_."A1.9.2"].ToteDir.toRight := FALSE;
	        END_IF;
	        
	    END_REGION
	    
	END_REGION
	
	REGION D1.1.1 Right
	    
	    IF IDB_ProductionLine."A1.9.1".CROSS_SENSOR_FILTER.SensorEdge.Negative AND
	        NOT IDB_ProductionLine."A1.9.1".CurrentPosition.right AND  //remobve not
	        NOT IDB_ProductionLine."A1.9.2".CurrentPosition.right //AND  // remove not
	        //NOT IDB_ProductionLine."D1.1.1".ReadConveyorStatus.Occupied
	    THEN
	        // Barcode
	        DB_ToteTracking.Conveyor[_."D1.1.1"].Barcode :=
	        DB_ToteTracking.Conveyor[_."A1.8.1"].Barcode;
	    END_IF;
	    
	END_REGION
	
	REGION D1.1.2
	    
	    IF IDB_ProductionLine."D1.1.1".CONVEYOR_SENSOR.SensorEdge.Negative THEN
	        DB_ToteTracking.Conveyor[_."D1.2.1"] := DB_ToteTracking.Conveyor[_."D1.1.1"];
	    END_IF;
	    
	END_REGION
	
	REGION D1.2.1
	    
	    IF IDB_ProductionLine."D1.2.1".CONVEYOR_SENSOR.SensorEdge.Negative THEN
	        DB_ToteTracking.Conveyor[_."D1.3.1"] := DB_ToteTracking.Conveyor[_."D1.2.1"];
	    END_IF;
	    
	END_REGION
	
	
	REGION A1.10.1 Straight
	    
	    IF IDB_ProductionLine."A1.9.1".CROSS_SENSOR_FILTER.SensorEdge.Negative AND
	        NOT IDB_ProductionLine."A1.9.1".CurrentPosition.straight AND  //remove not
	        NOT IDB_ProductionLine."A1.9.2".CurrentPosition.straight //AND  // remove not
	        //NOT IDB_ProductionLine."A1.10.1".ReadConveyorStatus.Occupied
	    THEN
	        // Barcode
	        DB_ToteTracking.Conveyor[_."A1.10.1"].Barcode :=
	        DB_ToteTracking.Conveyor[_."A1.8.1"].Barcode;
	    END_IF;
	    
	END_REGION
	
	REGION A1.10.2
	    
	    IF IDB_ProductionLine."A1.10.1".CONVEYOR_SENSOR.SensorEdge.Negative THEN
	        DB_ToteTracking.Conveyor[_."A1.10.2"] := DB_ToteTracking.Conveyor[_."A1.10.1"];
	    END_IF;
	    
	END_REGION
	
	REGION A1.10.3
	    
	    IF IDB_ProductionLine."A1.10.2".CONVEYOR_SENSOR.SensorEdge.Negative THEN
	        DB_ToteTracking.Conveyor[_."A1.10.3"] := DB_ToteTracking.Conveyor[_."A1.10.2"];
	    END_IF;
	    
	END_REGION
	
	
	
	
END_FUNCTION_BLOCK
END_NAMESPACE

NAMESPACE Global
FUNCTION_BLOCK FB_StatusON
{ S7_Optimized_Access := 'TRUE' ; Published := 'TRUE' }
VERSION : 0.1
   VAR_INPUT 
      SystemStartActive { ExternalAccessible := 'False'; ExternalVisible := 'False'; ExternalWritable := 'False'} : Bool;
      StatusStop { ExternalAccessible := 'False'; ExternalVisible := 'False'; ExternalWritable := 'False'} : Bool;
      StatusEStop { ExternalAccessible := 'False'; ExternalVisible := 'False'; ExternalWritable := 'False'} : Bool;
      StatusManual { ExternalAccessible := 'False'; ExternalVisible := 'False'; ExternalWritable := 'False'} : Bool;
      StatusFault { ExternalAccessible := 'False'; ExternalVisible := 'False'; ExternalWritable := 'False'} : Bool;
      FireAlarmActive { ExternalAccessible := 'False'; ExternalVisible := 'False'; ExternalWritable := 'False'} : Bool;
   END_VAR

   VAR_OUTPUT 
      StatusON { ExternalAccessible := 'False'; ExternalVisible := 'False'; ExternalWritable := 'False'} : Bool;
   END_VAR


BEGIN
	// ==========================================================================================================================================================================
	// Company       : LogTech, s.r.o.
	// Created by    : Anton Vinoth Soundraraj
	// Block         : FB_StatusON
	// Project       : LT-Lib-Block
	// ==========================================================================================================================================================================
	
	REGION STATUS ON
	    
	    IF #SystemStartActive AND NOT #StatusStop AND NOT #StatusEStop AND
	        NOT #StatusManual AND NOT #StatusFault AND NOT #FireAlarmActive
	    THEN
	        // The status of the conveyor is ON
	        #StatusON := TRUE;
	    END_IF;
	    
	    IF #StatusStop OR #StatusEStop OR #StatusManual OR
	        #StatusFault OR #FireAlarmActive THEN
	        // The status of the conveyor is OFF
	        #StatusON := FALSE;
	    END_IF;
	    
	END_REGION CONVEYOR STATUS ON
END_FUNCTION_BLOCK
END_NAMESPACE

DATA_BLOCK "FSIDB_Main_Safety_RTG1"   // DB1, F_DB
NAME : FUSI
// stored: InstanceOfName FSFB_Main_Safety_RTG1, InstanceOfType FB
"FSFB_Main_Safety_RTG1"
BEGIN
END_DATA_BLOCK

DATA_BLOCK "IDB_EmptyLine"   // DB9
// stored: InstanceOfName EmptyLine.FB_EmptyLine, InstanceOfType FB, Namespace EmptyLine
"EmptyLine.FB_EmptyLine"
   // VAR
   //    "J1.1.1" : "Global.FB_Conveyor";
   //    "J1.1.2" { S7_SetPoint := 'True'} : "Global.FB_Conveyor";
   //    "J1.1.3" { S7_SetPoint := 'True'} : "Global.FB_Conveyor";
   //    "J1.1.4" { S7_SetPoint := 'True'} : "Global.FB_Conveyor";
   //    "J1.1.5" { S7_SetPoint := 'True'} : "Global.FB_Conveyor";
   //    "J1.1.6" { S7_SetPoint := 'True'} : "Global.FB_Conveyor";
   //    "J1.1.7" { S7_SetPoint := 'True'} : "Global.FB_Conveyor";
   //    "J1.1.8" { S7_SetPoint := 'True'} : "Global.FB_Conveyor";
   //    "J1.1.9" { S7_SetPoint := 'True'} : "Global.FB_Conveyor";
   //    "J1.1.10" { S7_SetPoint := 'True'} : "Global.FB_Conveyor";
   //    "J1.1.11" { S7_SetPoint := 'True'} : "Global.FB_Conveyor";
   //    "J1.1.12" { S7_SetPoint := 'True'} : "Global.FB_Conveyor";
   //    "J1.1.13" { S7_SetPoint := 'True'} : "Global.FB_Conveyor";
   //    "J1.1.14" { S7_SetPoint := 'True'} : "Global.FB_Conveyor";
   //    "J1.1.15" { S7_SetPoint := 'True'} : "Global.FB_Conveyor";
   //    "J1.1.16" { S7_SetPoint := 'True'} : "Global.FB_Conveyor";
   //    "J1.2.1" { S7_SetPoint := 'True'} : "Global.FB_Conveyor";
   //    "J1.2.2" { S7_SetPoint := 'True'} : "Global.FB_Conveyor";
   //    "J1.2.3" { S7_SetPoint := 'True'} : "Global.FB_Conveyor";
   //    "J2.1.1" { S7_SetPoint := 'True'} : "Global.FB_Conveyor";
   //    "J2.1.2" { S7_SetPoint := 'True'} : "Global.FB_Conveyor";
   //    "J2.1.3" { S7_SetPoint := 'True'} : "Global.FB_Conveyor";
   //    "J2.1.4" { S7_SetPoint := 'True'} : "Global.FB_Conveyor";
   //    "J2.1.5" { S7_SetPoint := 'True'} : "Global.FB_Conveyor";
   //    "J2.1.6" { S7_SetPoint := 'True'} : "Global.FB_Conveyor";
   //    "J2.1.7" { S7_SetPoint := 'True'} : "Global.FB_Conveyor";
   //    "J2.1.8" { S7_SetPoint := 'True'} : "Global.FB_Conveyor";
   //    "J2.1.9" { S7_SetPoint := 'True'} : "Global.FB_Conveyor";
   //    "J2.1.10" { S7_SetPoint := 'True'} : "Global.FB_Conveyor";
   //    "J2.1.11" { S7_SetPoint := 'True'} : "Global.FB_Conveyor";
   //    "J2.1.12" { S7_SetPoint := 'True'} : "Global.FB_Conveyor";
   //    "J2.1.13" { S7_SetPoint := 'True'} : "Global.FB_Conveyor";
   //    "J2.1.14" { S7_SetPoint := 'True'} : "Global.FB_Conveyor";
   //    "J2.1.15" { S7_SetPoint := 'True'} : "Global.FB_Conveyor";
   //    "J2.2.1" { S7_SetPoint := 'True'} : "Global.FB_Conveyor";
   //    "J2.2.2" { S7_SetPoint := 'True'} : "Global.FB_Conveyor";
   //    "J2.3.1" { S7_SetPoint := 'True'} : "Global.FB_Conveyor";
   //    "J2.4.1" { S7_SetPoint := 'True'} : "Global.FB_Conveyor";
   //    "J1.2.4" { S7_SetPoint := 'True'} : "Global.FB_Conveyor";
   //    "J1.2.5" { S7_SetPoint := 'True'} : "Global.FB_Conveyor";
   //    "J1.3.1" { S7_SetPoint := 'True'} : "Global.FB_Conveyor";
   //    "J1.3.2" { S7_SetPoint := 'True'} : "Global.FB_Conveyor";
   //    "J1.4.1" { S7_SetPoint := 'True'} : "Global.FB_Conveyor";
   //    "J1.4.2" { S7_SetPoint := 'True'} : "Global.FB_Conveyor";
   //    "J1.4.3" { S7_SetPoint := 'True'} : "Global.FB_Conveyor";
   //    "J1.4.4" { S7_SetPoint := 'True'} : "Global.FB_Conveyor";
   //    "J1.4.5" { S7_SetPoint := 'True'} : "Global.FB_Conveyor";
   //    "J1.4.6" { S7_SetPoint := 'True'} : "Global.FB_Conveyor";
   //    "J1.4.7" { S7_SetPoint := 'True'} : "Global.FB_Conveyor";
   //    "J1.5.1" { S7_SetPoint := 'True'} : "Global.FB_Conveyor";
   //    "J1.5.2" { S7_SetPoint := 'True'} : "Global.FB_Conveyor";
   //    "J1.5.3" { S7_SetPoint := 'True'} : "Global.FB_Conveyor";
   //    "J1.5.4" { S7_SetPoint := 'True'} : "Global.FB_Conveyor";
   //    "J1.6.1" { S7_SetPoint := 'True'} : "Global.FB_MABS";
   //    "J1.6.2" { S7_SetPoint := 'True'} : "Global.FB_MABS";
   //    "J1.7.1" { S7_SetPoint := 'True'} : "Global.FB_Conveyor";
   //    "J1.7.2" { S7_SetPoint := 'True'} : "Global.FB_Conveyor";
   //    "J1.8.1" { S7_SetPoint := 'True'} : "Global.FB_Conveyor";
   //    "J1.8.2" { S7_SetPoint := 'True'} : "Global.FB_Conveyor";
   //    "J1.9.1" { S7_SetPoint := 'True'} : "Global.FB_Conveyor";
   //    "J1.10.1" { S7_SetPoint := 'True'} : "Global.FB_Conveyor";
   //    "J1.11.1" { S7_SetPoint := 'True'} : "Global.FB_Conveyor";
   //    "J1.11.2" { S7_SetPoint := 'True'} : "Global.FB_Conveyor";
   //    "J1.11.3" { S7_SetPoint := 'True'} : "Global.FB_Conveyor";
   //    "J1.11.4" { S7_SetPoint := 'True'} : "Global.FB_Conveyor";
   //    "J1.11.5" { S7_SetPoint := 'True'} : "Global.FB_Conveyor";
   //    "J1.11.6" { S7_SetPoint := 'True'} : "Global.FB_Conveyor";
   //    "J1.11.7" { S7_SetPoint := 'True'} : "Global.FB_Conveyor";
   //    "J1.11.8" { S7_SetPoint := 'True'} : "Global.FB_Conveyor";
   //    "J1.11.9" { S7_SetPoint := 'True'} : "Global.FB_Conveyor";
   //    "J1.11.10" { S7_SetPoint := 'True'} : "Global.FB_Conveyor";
   //    "J1.11.11" { S7_SetPoint := 'True'} : "Global.FB_Conveyor";
   //    "J1.11.12" { S7_SetPoint := 'True'} : "Global.FB_Conveyor";
   //    "J1.11.13" { S7_SetPoint := 'True'} : "Global.FB_Conveyor";
   //    "K1.1.1" { S7_SetPoint := 'True'} : "Global.FB_Conveyor";
   //    "K1.2.1" { S7_SetPoint := 'True'} : "Global.FB_Conveyor";
   //    "K1.3.1" { S7_SetPoint := 'True'} : "Global.FB_Conveyor";
   //    "K1.4.1" { S7_SetPoint := 'True'} : "Global.FB_Conveyor";
   //    "K1.4.2" { S7_SetPoint := 'True'} : "Global.FB_Conveyor";
   //    "K1.4.3" { S7_SetPoint := 'True'} : "Global.FB_Conveyor";
   //    "K1.4.4" { S7_SetPoint := 'True'} : "Global.FB_Conveyor";
   //    "K1.4.5" { S7_SetPoint := 'True'} : "Global.FB_Conveyor";
   //    "K1.4.6" { S7_SetPoint := 'True'} : "Global.FB_Conveyor";
   //    "K1.4.7" { S7_SetPoint := 'True'} : "Global.FB_Conveyor";
   //    "K1.4.8" { S7_SetPoint := 'True'} : "Global.FB_Conveyor";
   //    "K1.4.9" { S7_SetPoint := 'True'} : "Global.FB_Conveyor";
   //    "K1.4.10" { S7_SetPoint := 'True'} : "Global.FB_Conveyor";
   //    "K1.5.1" { S7_SetPoint := 'True'} : "Global.FB_Conveyor";
   //    "K1.5.2" { S7_SetPoint := 'True'} : "Global.FB_Conveyor";
   //    "K1.5.3" { S7_SetPoint := 'True'} : "Global.FB_Conveyor";
   //    "K1.5.4" { S7_SetPoint := 'True'} : "Global.FB_Conveyor";
   //    "K1.5.5" { S7_SetPoint := 'True'} : "Global.FB_Conveyor";
   //    "K1.5.6" { S7_SetPoint := 'True'} : "Global.FB_Conveyor";
   //    "K1.5.7" { S7_SetPoint := 'True'} : "Global.FB_Conveyor";
   //    "K1.5.8" { S7_SetPoint := 'True'} : "Global.FB_Conveyor";
   //    "K1.6.1" { S7_SetPoint := 'True'} : "Global.FB_Conveyor";
   //    "K1.6.2" { S7_SetPoint := 'True'} : "Global.FB_Conveyor";
   //    "K1.7.1" { S7_SetPoint := 'True'} : "Global.FB_Conveyor";
   //    "K1.7.2" { S7_SetPoint := 'True'} : "Global.FB_Conveyor";
   //    "K1.8.1" { S7_SetPoint := 'True'} : "Global.FB_Conveyor";
   //    "K1.8.2" { S7_SetPoint := 'True'} : "Global.FB_Conveyor";
   //    "K1.8.3" { S7_SetPoint := 'True'} : "Global.FB_Conveyor";
   //    "K1.9.1" { S7_SetPoint := 'True'} : "Global.FB_Conveyor";
   //    "K1.9.2" { S7_SetPoint := 'True'} : "Global.FB_Conveyor";
   //    "K1.9.3" { S7_SetPoint := 'True'} : "Global.FB_Conveyor";
   //    "K1.9.4" { S7_SetPoint := 'True'} : "Global.FB_Conveyor";
   //    "K1.9.5" { S7_SetPoint := 'True'} : "Global.FB_Conveyor";
   //    "K1.9.6" { S7_SetPoint := 'True'} : "Global.FB_Conveyor";
   //    "K1.9.7" { S7_SetPoint := 'True'} : "Global.FB_Conveyor";
   //    "K1.10.1" { S7_SetPoint := 'True'} : "Global.FB_Conveyor";
   // END_VAR
BEGIN
END_DATA_BLOCK

DATA_BLOCK "IDB_GlobalStatus"   // DB48
// stored: InstanceOfName Global.FB_GlobalStatus, InstanceOfType FB, Namespace Global
"Global.FB_GlobalStatus"
   // VAR
   //    Line : Struct
   //       ProductionLine : "Global.ConveyorStatus";
   //       EmptyLine { S7_SetPoint := 'True'} : "Global.ConveyorStatus";
   //       PackedLine { S7_SetPoint := 'True'} : "Global.ConveyorStatus";
   //    END_STRUCT;
   //    cmp : Struct
   //       ProductionTotes_Value0 : Array[_.gminProductionLine.._.gmaxProductionLine] of Bool;
   //       ProductionTotes_Value1 : Array[_.gminProductionLine.._.gmaxProductionLine] of Bool;
   //       EmptyLine_Value0 : Array[_.gminEmptyLine.._.gmaxEmptyLine] of Bool;
   //       EmptyLine_Value1 : Array[_.gminEmptyLine.._.gmaxEmptyLine] of Bool;
   //       PackedLine_Value0 : Array[_.gminPackedLine.._.gmaxPackedLine] of Bool;
   //       PackedLine_Value1 : Array[_.gminPackedLine.._.gmaxPackedLine] of Bool;
   //    END_STRUCT;
   //    ForVisu : Struct
   //       Line : Struct
   //          ProductionLine : Word;
   //          EmptyLine : Word;
   //          PackedLine : Word;
   //       END_STRUCT;
   //    END_STRUCT;
   // END_VAR
BEGIN
   cmp.ProductionTotes_Value1[1001..1192] := True;
   cmp.EmptyLine_Value1[2001..2109] := True;
   cmp.PackedLine_Value1[3001..3040] := True;
END_DATA_BLOCK

DATA_BLOCK "IDB_PackedLine"   // DB10
// stored: Access Published, InstanceOfName PackedLine.FB_PackedLine, InstanceOfType FB, Namespace PackedLine
"PackedLine.FB_PackedLine"
   // VAR
   //    "G1.1.1" { S7_SetPoint := 'True'} : "Global.FB_Conveyor";
   //    "G1.1.2" { S7_SetPoint := 'True'} : "Global.FB_Conveyor";
   //    "G1.1.3" { S7_SetPoint := 'True'} : "Global.FB_Conveyor";
   //    "G1.1.4" { S7_SetPoint := 'True'} : "Global.FB_Conveyor";
   //    "G1.1.5" { S7_SetPoint := 'True'} : "Global.FB_Conveyor";
   //    "G1.1.6" { S7_SetPoint := 'True'} : "Global.FB_Conveyor";
   //    "G1.1.7" { S7_SetPoint := 'True'} : "Global.FB_Conveyor";
   //    "G1.1.8" { S7_SetPoint := 'True'} : "Global.FB_Conveyor";
   //    "G1.1.9" { S7_SetPoint := 'True'} : "Global.FB_Conveyor";
   //    "G1.1.10" { S7_SetPoint := 'True'} : "Global.FB_Conveyor";
   //    "G1.1.11" { S7_SetPoint := 'True'} : "Global.FB_Conveyor";
   //    "G1.1.12" { S7_SetPoint := 'True'} : "Global.FB_Conveyor";
   //    "G1.1.13" { S7_SetPoint := 'True'} : "Global.FB_Conveyor";
   //    "G1.1.14" { S7_SetPoint := 'True'} : "Global.FB_Conveyor";
   //    "G1.1.15" { S7_SetPoint := 'True'} : "Global.FB_Conveyor";
   //    "G1.1.16" { S7_SetPoint := 'True'} : "Global.FB_Conveyor";
   //    "G1.1.17" { S7_SetPoint := 'True'} : "Global.FB_Conveyor";
   //    "G1.1.18" { S7_SetPoint := 'True'} : "Global.FB_Conveyor";
   //    "G1.1.19" { S7_SetPoint := 'True'} : "Global.FB_Conveyor";
   //    "G1.2.1" { S7_SetPoint := 'True'} : "Global.FB_Conveyor";
   //    "G1.2.2" { S7_SetPoint := 'True'} : "Global.FB_Conveyor";
   //    "G1.3.1" { S7_SetPoint := 'True'} : "Global.FB_Conveyor";
   //    "G1.4.1" { S7_SetPoint := 'True'} : "Global.FB_Conveyor";
   //    "G1.4.2" { S7_SetPoint := 'True'} : "Global.FB_Conveyor";
   //    "G1.4.3" { S7_SetPoint := 'True'} : "Global.FB_Conveyor";
   //    "G1.4.4" { S7_SetPoint := 'True'} : "Global.FB_Conveyor";
   //    "G1.4.5" { S7_SetPoint := 'True'} : "Global.FB_Conveyor";
   //    "G1.4.6" { S7_SetPoint := 'True'} : "Global.FB_Conveyor";
   //    "G1.5.1" { S7_SetPoint := 'True'} : "Global.FB_Conveyor";
   //    "G1.5.2" { S7_SetPoint := 'True'} : "Global.FB_Conveyor";
   //    "G1.5.3" { S7_SetPoint := 'True'} : "Global.FB_Conveyor";
   //    "G1.5.4" { S7_SetPoint := 'True'} : "Global.FB_Conveyor";
   //    "G1.5.5" { S7_SetPoint := 'True'} : "Global.FB_Conveyor";
   //    "G1.5.6" { S7_SetPoint := 'True'} : "Global.FB_Conveyor";
   //    "G1.6.1" { S7_SetPoint := 'True'} : "Global.FB_Conveyor";
   //    "G1.6.2" { S7_SetPoint := 'True'} : "Global.FB_Conveyor";
   //    "G1.7.1" { S7_SetPoint := 'True'} : "Global.FB_Conveyor";
   //    "G1.7.2" { S7_SetPoint := 'True'} : "Global.FB_Conveyor";
   //    "G1.7.3" { S7_SetPoint := 'True'} : "Global.FB_Conveyor";
   //    "G1.7.4" { S7_SetPoint := 'True'} : "Global.FB_Conveyor";
   // END_VAR
BEGIN
END_DATA_BLOCK

DATA_BLOCK "IDB_Merging"   // DB27
// stored: InstanceOfName ProductionLine.FB_Merging, InstanceOfType FB, Namespace ProductionLine
"ProductionLine.FB_Merging"
   // VAR
   //    "Merge_A1.7.3" : "Global.FB_Merging";
   //    "Merge_A1.9.3" : "Global.FB_Merging";
   //    "Merge_B1.6.1" { S7_SetPoint := 'True'} : "Global.FB_Merging";
   // END_VAR
BEGIN
END_DATA_BLOCK

DATA_BLOCK "IDB_ProductionLine"   // DB8
// stored: InstanceOfName ProductionLine.FB_ProductionLine, InstanceOfType FB, Namespace ProductionLine
"ProductionLine.FB_ProductionLine"
   // VAR
   //    "A1.1.1" { S7_SetPoint := 'True'} : "Global.FB_Conveyor";
   //    "A1.1.2" { S7_SetPoint := 'True'} : "Global.FB_Conveyor";
   //    "A1.1.3" { S7_SetPoint := 'True'} : "Global.FB_Conveyor";
   //    "A1.1.4" { S7_SetPoint := 'True'} : "Global.FB_Conveyor";
   //    "A1.1.5" { S7_SetPoint := 'True'} : "Global.FB_Conveyor";
   //    "A1.1.6" { S7_SetPoint := 'True'} : "Global.FB_Conveyor";
   //    "A1.1.7" { S7_SetPoint := 'True'} : "Global.FB_Conveyor";
   //    "A1.1.8" { S7_SetPoint := 'True'} : "Global.FB_Conveyor";
   //    "A1.1.9" { S7_SetPoint := 'True'} : "Global.FB_Conveyor";
   //    "A1.1.10" { S7_SetPoint := 'True'} : "Global.FB_Conveyor";
   //    "A1.1.11" { S7_SetPoint := 'True'} : "Global.FB_Conveyor";
   //    "A1.1.12" { S7_SetPoint := 'True'} : "Global.FB_Conveyor";
   //    "A1.1.13" { S7_SetPoint := 'True'} : "Global.FB_Conveyor";
   //    "A1.1.14" { S7_SetPoint := 'True'} : "Global.FB_Conveyor";
   //    "A1.2.1" { S7_SetPoint := 'True'} : "Global.FB_Conveyor";
   //    "A1.3.1" { S7_SetPoint := 'True'} : "Global.FB_Conveyor";
   //    "A1.4.1" { S7_SetPoint := 'True'} : "Global.FB_Conveyor";
   //    "A1.5.1" { S7_SetPoint := 'True'} : "Global.FB_Conveyor";
   //    "A1.5.2" { S7_SetPoint := 'True'} : "Global.FB_Conveyor";
   //    "A1.5.3" { S7_SetPoint := 'True'} : "Global.FB_Conveyor";
   //    "A1.7.1" { S7_SetPoint := 'True'} : "Global.FB_Conveyor";
   //    "A1.7.2" { S7_SetPoint := 'True'} : "Global.FB_Conveyor";
   //    "A1.7.3" { S7_SetPoint := 'True'} : "Global.FB_Conveyor";
   //    "A1.7.4" { S7_SetPoint := 'True'} : "Global.FB_Conveyor";
   //    "A1.7.5" { S7_SetPoint := 'True'} : "Global.FB_Conveyor";
   //    "A1.7.6" { S7_SetPoint := 'True'} : "Global.FB_Conveyor";
   //    "A1.8.1" { S7_SetPoint := 'True'} : "Global.FB_Conveyor";
   //    "A1.10.1" { S7_SetPoint := 'True'} : "Global.FB_Conveyor";
   //    "A1.10.2" { S7_SetPoint := 'True'} : "Global.FB_Conveyor";
   //    "A1.10.3" { S7_SetPoint := 'True'} : "Global.FB_Conveyor";
   //    "A1.10.4" { S7_SetPoint := 'True'} : "Global.FB_Conveyor";
   //    "A1.10.5" { S7_SetPoint := 'True'} : "Global.FB_Conveyor";
   //    "A1.10.6" { S7_SetPoint := 'True'} : "Global.FB_Conveyor";
   //    "A1.10.7" { S7_SetPoint := 'True'} : "Global.FB_Conveyor";
   //    "A1.10.8" { S7_SetPoint := 'True'} : "Global.FB_Conveyor";
   //    "A1.10.9" { S7_SetPoint := 'True'} : "Global.FB_Conveyor";
   //    "A1.10.10" { S7_SetPoint := 'True'} : "Global.FB_Conveyor";
   //    "A1.10.11" { S7_SetPoint := 'True'} : "Global.FB_Conveyor";
   //    "A1.10.12" { S7_SetPoint := 'True'} : "Global.FB_Conveyor";
   //    "A1.10.13" { S7_SetPoint := 'True'} : "Global.FB_Conveyor";
   //    "A1.11.1" { S7_SetPoint := 'True'} : "Global.FB_Conveyor";
   //    "A1.11.2" { S7_SetPoint := 'True'} : "Global.FB_Conveyor";
   //    "A1.12.1" { S7_SetPoint := 'True'} : "Global.FB_Conveyor";
   //    "A1.12.2" { S7_SetPoint := 'True'} : "Global.FB_Conveyor";
   //    "A1.14.1" { S7_SetPoint := 'True'} : "Global.FB_Conveyor";
   //    "A1.14.2" { S7_SetPoint := 'True'} : "Global.FB_Conveyor";
   //    "A1.14.3" { S7_SetPoint := 'True'} : "Global.FB_Conveyor";
   //    "A1.14.4" { S7_SetPoint := 'True'} : "Global.FB_Conveyor";
   //    "A1.14.5" { S7_SetPoint := 'True'} : "Global.FB_Conveyor";
   //    "A1.14.6" { S7_SetPoint := 'True'} : "Global.FB_Conveyor";
   //    "A1.14.7" { S7_SetPoint := 'True'} : "Global.FB_Conveyor";
   //    "A1.14.8" { S7_SetPoint := 'True'} : "Global.FB_Conveyor";
   //    "A1.14.9" { S7_SetPoint := 'True'} : "Global.FB_Conveyor";
   //    "A1.14.10" { S7_SetPoint := 'True'} : "Global.FB_Conveyor";
   //    "A1.14.11" { S7_SetPoint := 'True'} : "Global.FB_Conveyor";
   //    "A1.14.12" { S7_SetPoint := 'True'} : "Global.FB_Conveyor";
   //    "A1.14.13" { S7_SetPoint := 'True'} : "Global.FB_Conveyor";
   //    "A1.14.14" { S7_SetPoint := 'True'} : "Global.FB_Conveyor";
   //    "A1.14.15" { S7_SetPoint := 'True'} : "Global.FB_Conveyor";
   //    "A1.14.16" { S7_SetPoint := 'True'} : "Global.FB_Conveyor";
   //    "A1.14.17" { S7_SetPoint := 'True'} : "Global.FB_Conveyor";
   //    "A1.14.18" { S7_SetPoint := 'True'} : "Global.FB_Conveyor";
   //    "A1.14.19" { S7_SetPoint := 'True'} : "Global.FB_Conveyor";
   //    "A1.14.20" { S7_SetPoint := 'True'} : "Global.FB_Conveyor";
   //    "A1.14.21" { S7_SetPoint := 'True'} : "Global.FB_Conveyor";
   //    "A1.14.22" { S7_SetPoint := 'True'} : "Global.FB_Conveyor";
   //    "A1.14.23" { S7_SetPoint := 'True'} : "Global.FB_Conveyor";
   //    "A1.14.24" { S7_SetPoint := 'True'} : "Global.FB_Conveyor";
   //    "A1.14.25" { S7_SetPoint := 'True'} : "Global.FB_Conveyor";
   //    "A1.14.26" { S7_SetPoint := 'True'} : "Global.FB_Conveyor";
   //    "A2.2.1" { S7_SetPoint := 'True'} : "Global.FB_Conveyor";
   //    "A2.2.2" { S7_SetPoint := 'True'} : "Global.FB_Conveyor";
   //    "A2.2.3" { S7_SetPoint := 'True'} : "Global.FB_Conveyor";
   //    "A2.2.4" { S7_SetPoint := 'True'} : "Global.FB_Conveyor";
   //    "A2.2.5" { S7_SetPoint := 'True'} : "Global.FB_Conveyor";
   //    "A2.2.6" { S7_SetPoint := 'True'} : "Global.FB_Conveyor";
   //    "A2.2.7" { S7_SetPoint := 'True'} : "Global.FB_Conveyor";
   //    "A2.2.8" { S7_SetPoint := 'True'} : "Global.FB_Conveyor";
   //    "A2.2.9" { S7_SetPoint := 'True'} : "Global.FB_Conveyor";
   //    "A2.2.10" { S7_SetPoint := 'True'} : "Global.FB_Conveyor";
   //    "A2.2.11" { S7_SetPoint := 'True'} : "Global.FB_Conveyor";
   //    "A2.2.12" { S7_SetPoint := 'True'} : "Global.FB_Conveyor";
   //    "A2.2.13" { S7_SetPoint := 'True'} : "Global.FB_Conveyor";
   //    "A2.2.14" { S7_SetPoint := 'True'} : "Global.FB_Conveyor";
   //    "A2.2.15" { S7_SetPoint := 'True'} : "Global.FB_Conveyor";
   //    "A2.2.16" { S7_SetPoint := 'True'} : "Global.FB_Conveyor";
   //    "A2.2.17" { S7_SetPoint := 'True'} : "Global.FB_Conveyor";
   //    "A2.2.18" { S7_SetPoint := 'True'} : "Global.FB_Conveyor";
   //    "A2.2.19" { S7_SetPoint := 'True'} : "Global.FB_Conveyor";
   //    "A2.2.20" { S7_SetPoint := 'True'} : "Global.FB_Conveyor";
   //    "A2.2.21" { S7_SetPoint := 'True'} : "Global.FB_Conveyor";
   //    "A2.2.22" { S7_SetPoint := 'True'} : "Global.FB_Conveyor";
   //    "A2.2.23" { S7_SetPoint := 'True'} : "Global.FB_Conveyor";
   //    "A2.2.24" { S7_SetPoint := 'True'} : "Global.FB_Conveyor";
   //    "A2.2.25" { S7_SetPoint := 'True'} : "Global.FB_Conveyor";
   //    "A2.2.26" { S7_SetPoint := 'True'} : "Global.FB_Conveyor";
   //    "B1.1.1" { S7_SetPoint := 'True'} : "Global.FB_Conveyor";
   //    "B1.2.1" { S7_SetPoint := 'True'} : "Global.FB_Conveyor";
   //    "B1.3.1" { S7_SetPoint := 'True'} : "Global.FB_Conveyor";
   //    "B1.3.2" { S7_SetPoint := 'True'} : "Global.FB_Conveyor";
   //    "B1.3.3" { S7_SetPoint := 'True'} : "Global.FB_Conveyor";
   //    "B1.4.1" { S7_SetPoint := 'True'} : "Global.FB_Conveyor";
   //    "B1.4.2" { S7_SetPoint := 'True'} : "Global.FB_Conveyor";
   //    "B1.5.1" { S7_SetPoint := 'True'} : "Global.FB_Conveyor";
   //    "B1.7.1" { S7_SetPoint := 'True'} : "Global.FB_Conveyor";
   //    "B1.7.2" { S7_SetPoint := 'True'} : "Global.FB_Conveyor";
   //    "B1.7.3" { S7_SetPoint := 'True'} : "Global.FB_Conveyor";
   //    "B1.8.1" { S7_SetPoint := 'True'} : "Global.FB_Conveyor";
   //    "B1.8.2" { S7_SetPoint := 'True'} : "Global.FB_Conveyor";
   //    "B1.8.3" { S7_SetPoint := 'True'} : "Global.FB_Conveyor";
   //    "B1.9.1" { S7_SetPoint := 'True'} : "Global.FB_Conveyor";
   //    "B1.9.2" { S7_SetPoint := 'True'} : "Global.FB_Conveyor";
   //    "B1.11.1" { S7_SetPoint := 'True'} : "Global.FB_Conveyor";
   //    "B1.11.2" { S7_SetPoint := 'True'} : "Global.FB_Conveyor";
   //    "B1.11.3" { S7_SetPoint := 'True'} : "Global.FB_Conveyor";
   //    "B1.11.4" { S7_SetPoint := 'True'} : "Global.FB_Conveyor";
   //    "B1.12.1" { S7_SetPoint := 'True'} : "Global.FB_Conveyor";
   //    "B1.12.2" { S7_SetPoint := 'True'} : "Global.FB_Conveyor";
   //    "B1.15.1" { S7_SetPoint := 'True'} : "Global.FB_Conveyor";
   //    "B1.15.2" { S7_SetPoint := 'True'} : "Global.FB_Conveyor";
   //    "B1.16.1" { S7_SetPoint := 'True'} : "Global.FB_Conveyor";
   //    "B1.16.2" { S7_SetPoint := 'True'} : "Global.FB_Conveyor";
   //    "B1.16.3" { S7_SetPoint := 'True'} : "Global.FB_Conveyor";
   //    "B1.16.4" { S7_SetPoint := 'True'} : "Global.FB_Conveyor";
   //    "B1.16.5" { S7_SetPoint := 'True'} : "Global.FB_Conveyor";
   //    "B1.16.6" { S7_SetPoint := 'True'} : "Global.FB_Conveyor";
   //    "B1.16.7" { S7_SetPoint := 'True'} : "Global.FB_Conveyor";
   //    "B1.16.8" { S7_SetPoint := 'True'} : "Global.FB_Conveyor";
   //    "B1.17.1" { S7_SetPoint := 'True'} : "Global.FB_Conveyor";
   //    "B1.17.2" { S7_SetPoint := 'True'} : "Global.FB_Conveyor";
   //    "B1.17.3" { S7_SetPoint := 'True'} : "Global.FB_Conveyor";
   //    "B1.17.4" { S7_SetPoint := 'True'} : "Global.FB_Conveyor";
   //    "B1.19.1" { S7_SetPoint := 'True'} : "Global.FB_Conveyor";
   //    "B1.20.1" { S7_SetPoint := 'True'} : "Global.FB_Conveyor";
   //    "B1.20.2" { S7_SetPoint := 'True'} : "Global.FB_Conveyor";
   //    "B1.21.1" { S7_SetPoint := 'True'} : "Global.FB_Conveyor";
   //    "B1.21.2" { S7_SetPoint := 'True'} : "Global.FB_Conveyor";
   //    "B1.21.3" { S7_SetPoint := 'True'} : "Global.FB_Conveyor";
   //    "B1.22.1" { S7_SetPoint := 'True'} : "Global.FB_Conveyor";
   //    "B1.23.1" { S7_SetPoint := 'True'} : "Global.FB_Conveyor";
   //    "C1.2.2" { S7_SetPoint := 'True'} : "Global.FB_Conveyor";
   //    "C1.2.1" { S7_SetPoint := 'True'} : "Global.FB_Conveyor";
   //    "C1.4.1" { S7_SetPoint := 'True'} : "Global.FB_Conveyor";
   //    "C1.4.2" { S7_SetPoint := 'True'} : "Global.FB_Conveyor";
   //    "D1.1.1" { S7_SetPoint := 'True'} : "Global.FB_Conveyor";
   //    "D1.2.1" { S7_SetPoint := 'True'} : "Global.FB_Conveyor";
   //    "D1.3.1" { S7_SetPoint := 'True'} : "Global.FB_Conveyor";
   //    "D1.4.1" { S7_SetPoint := 'True'} : "Global.FB_Conveyor";
   //    "D1.5.1" { S7_SetPoint := 'True'} : "Global.FB_Conveyor";
   //    "D1.6.1" { S7_SetPoint := 'True'} : "Global.FB_Conveyor";
   //    "D1.7.1" { S7_SetPoint := 'True'} : "Global.FB_Conveyor";
   //    "D1.7.2" { S7_SetPoint := 'True'} : "Global.FB_Conveyor";
   //    "D1.7.3" { S7_SetPoint := 'True'} : "Global.FB_Conveyor";
   //    "D1.7.4" { S7_SetPoint := 'True'} : "Global.FB_Conveyor";
   //    "D1.7.5" { S7_SetPoint := 'True'} : "Global.FB_Conveyor";
   //    "D1.7.6" { S7_SetPoint := 'True'} : "Global.FB_Conveyor";
   //    "D1.7.7" { S7_SetPoint := 'True'} : "Global.FB_Conveyor";
   //    "D1.7.8" { S7_SetPoint := 'True'} : "Global.FB_Conveyor";
   //    "D1.7.9" { S7_SetPoint := 'True'} : "Global.FB_Conveyor";
   //    "D1.7.10" { S7_SetPoint := 'True'} : "Global.FB_Conveyor";
   //    "D1.8.1" { S7_SetPoint := 'True'} : "Global.FB_Conveyor";
   //    "D1.8.2" { S7_SetPoint := 'True'} : "Global.FB_Conveyor";
   //    "D1.8.3" { S7_SetPoint := 'True'} : "Global.FB_Conveyor";
   //    "D1.11.1" { S7_SetPoint := 'True'} : "Global.FB_Conveyor";
   //    "D1.11.2" { S7_SetPoint := 'True'} : "Global.FB_Conveyor";
   //    "D1.11.3" { S7_SetPoint := 'True'} : "Global.FB_Conveyor";
   //    "D1.12.1" { S7_SetPoint := 'True'} : "Global.FB_Conveyor";
   //    "D1.12.2" { S7_SetPoint := 'True'} : "Global.FB_Conveyor";
   //    "D1.12.3" { S7_SetPoint := 'True'} : "Global.FB_Conveyor";
   //    "E1.1.1" { S7_SetPoint := 'True'} : "Global.FB_Conveyor";
   //    "E1.1.2" { S7_SetPoint := 'True'} : "Global.FB_Conveyor";
   //    "E1.1.3" { S7_SetPoint := 'True'} : "Global.FB_Conveyor";
   //    "E1.1.4" { S7_SetPoint := 'True'} : "Global.FB_Conveyor";
   //    "E1.2.1" { S7_SetPoint := 'True'} : "Global.FB_Conveyor";
   //    "E1.3.1" { S7_SetPoint := 'True'} : "Global.FB_Conveyor";
   //    "E1.4.1" { S7_SetPoint := 'True'} : "Global.FB_Conveyor";
   //    "E1.5.1" { S7_SetPoint := 'True'} : "Global.FB_Conveyor";
   //    "E1.6.1" { S7_SetPoint := 'True'} : "Global.FB_Conveyor";
   //    "A1.9.1" { S7_SetPoint := 'True'} : "Global.FB_MABS";
   //    "A1.9.2" { S7_SetPoint := 'True'} : "Global.FB_MABS";
   //    "A1.6.1" { S7_SetPoint := 'True'} : "Global.FB_MABS";
   //    "A1.6.2" { S7_SetPoint := 'True'} : "Global.FB_MABS";
   //    "A1.13.1" { S7_SetPoint := 'True'} : "Global.FB_S300_tTransMode";
   //    "A2.1.1" { S7_SetPoint := 'True'} : "Global.FB_S300_tTransMode";
   //    "B1.6.1" { S7_SetPoint := 'True'} : "Global.FB_S300_FullControl";
   //    "B1.10.1" { S7_SetPoint := 'True'} : "Global.FB_S300_tTransMode";
   //    "B1.13.1" { S7_SetPoint := 'True'} : "Global.FB_S300_tTransMode";
   //    "B1.14.1" { S7_SetPoint := 'True'} : "Global.FB_S300_tTransMode";
   //    "B1.18.1" { S7_SetPoint := 'True'} : "Global.FB_S300_tTransMode";
   //    "C1.3.1" { S7_SetPoint := 'True'} : "Global.FB_S300_tTransMode";
   //    "D1.9.2" { S7_SetPoint := 'True'} : "Global.FB_S300_tTransMode";
   //    "D1.10.1" { S7_SetPoint := 'True'} : "Global.FB_S300_tTransMode";
   // END_VAR
BEGIN
END_DATA_BLOCK

DATA_BLOCK "IDB_HardwareDiag"   // DB12
// stored: Access Published, InstanceOfName Global.FB_HardwareDiag, InstanceOfType FB, Namespace Global
"Global.FB_HardwareDiag"
   // VAR
   //    "BW-ASi -10.106.129.143" : "Global.FB_GetDiag";
   //    "BW-ASi -10.106.129.200" { S7_SetPoint := 'True'} : "Global.FB_GetDiag";
   //    "Cognex -10.106.129.24" : "Global.FB_GetDiag";
   //    "Cognex -10.106.129.25" { S7_SetPoint := 'True'} : "Global.FB_GetDiag";
   //    "Cognex -10.106.129.26" { S7_SetPoint := 'True'} : "Global.FB_GetDiag";
   //    "Cognex -10.106.129.27" { S7_SetPoint := 'True'} : "Global.FB_GetDiag";
   //    "IMC - 10.106.129.84" { S7_SetPoint := 'True'} : "Global.FB_GetDiag";
   //    "IMC - 10.106.129.85" { S7_SetPoint := 'True'} : "Global.FB_GetDiag";
   //    "IMC - 10.106.129.86" { S7_SetPoint := 'True'} : "Global.FB_GetDiag";
   //    "IMC - 10.106.129.87" { S7_SetPoint := 'True'} : "Global.FB_GetDiag";
   //    "IMC - 10.106.129.88" { S7_SetPoint := 'True'} : "Global.FB_GetDiag";
   // END_VAR
BEGIN
END_DATA_BLOCK

DATA_BLOCK "IDB_VisuAlarm"   // DB49
// stored: Access Published, InstanceOfName Global.FB_VisuAlarm, InstanceOfType FB, Namespace Global
"Global.FB_VisuAlarm"
   // VAR
   //    noAlarmState : Bool;
   //    CommunicationFault : Struct
   //       PLC : Word;
   //       "BW-ASi" : Word;
   //       Cognex : Word;
   //       Mabs : Word;
   //    END_STRUCT;
   //    "BW-ASi" : Struct
   //       "BW_ASi143 -MCC100 -210KE3 -ConfigErr_Circuit1_Slave(0-15)A_1" : Word;
   //       "BW_ASi143 -MCC100 -210KE3 -ConfigErr_Circuit1_Slave(16-31)A" : Word;
   //       "BW_ASi143 -MCC100 -210KE3 -ConfigErr_Circuit1_Slave(0-15)B_1" : Word;
   //       "BW_ASi143 -MCC100 -210KE3 -ConfigErr_Circuit1_Slave(16-31)B" : Word;
   //       "BW_ASi143 -MCC100 -210KE3 -PeriErr_Circuit1_Slave(0-15)A_1" : Word;
   //       "BW_ASi143 -MCC100 -210KE3 -PeriErr_Circuit1_Slave(16-31)A" : Word;
   //       "BW_ASi143 -MCC100 -210KE3 -PeriErr_Circuit1_Slave(0-15)B_1" : Word;
   //       "BW_ASi143 -MCC100 -210KE3 -PeriErr_Circuit1_Slave(16-31)B" : Word;
   //       "BW_ASi143 -MCC100 -210KE3 -ConfigErr_Circuit2_Slave(0-15)A" : Word;
   //       "BW_ASi143 -MCC100 -210KE3 -ConfigErr_Circuit2_Slave(16-31)A" : Word;
   //       "BW_ASi143 -MCC100 -210KE3 -ConfigErr_Circuit2_Slave(0-15)B" : Word;
   //       "BW_ASi143 -MCC100 -210KE3 -ConfigErr_Circuit2_Slave(16-31)B" : Word;
   //       "BW_ASi143 -MCC100 -210KE3 -PeriErr_Circuit2_Slave(0-15)A" : Word;
   //       "BW_ASi143 -MCC100 -210KE3 -PeriErr_Circuit2_Slave(16-31)A" : Word;
   //       "BW_ASi143 -MCC100 -210KE3 -PeriErr_Circuit2_Slave(0-15)B" : Word;
   //       "BW_ASi143 -MCC100 -210KE3 -PeriErr_Circuit2_Slave(16-31)B" : Word;
   //       "BW_ASi200 -MCC300 -210KE3 -ConfigErr_Circuit1_Slave(0-15)A" : Word;
   //       "BW_ASi200 -MCC300 -210KE3 -ConfigErr_Circuit1_Slave(16-31)A" : Word;
   //       "BW_ASi200 -MCC300 -210KE3 -ConfigErr_Circuit1_Slave(0-15)B" : Word;
   //       "BW_ASi200 -MCC300 -210KE3 -ConfigErr_Circuit1_Slave(16-31)B" : Word;
   //       "BW_ASi200 -MCC300 -210KE3 -PeriErr_Circuit1_Slave(0-15)A" : Word;
   //       "BW_ASi200 -MCC300 -210KE3 -PeriErr_Circuit1_Slave(16-31)A" : Word;
   //       "BW_ASi200 -MCC300 -210KE3 -PeriErr_Circuit1_Slave(0-15)B" : Word;
   //       "BW_ASi200 -MCC300 -210KE3 -PeriErr_Circuit1_Slave(16-31)B" : Word;
   //       "BW_ASi200 -MCC300 -210KE3 -ConfigErr_Circuit2_Slave(0-15)A" : Word;
   //       "BW_ASi200 -MCC300 -210KE3 -ConfigErr_Circuit2_Slave(16-31)A" : Word;
   //       "BW_ASi200 -MCC300 -210KE3 -ConfigErr_Circuit2_Slave(0-15)B" : Word;
   //       "BW_ASi200 -MCC300 -210KE3 -ConfigErr_Circuit2_Slave(16-31)B" : Word;
   //       "BW_ASi200 -MCC300 -210KE3 -PeriErr_Circuit2_Slave(0-15)A" : Word;
   //       "BW_ASi200 -MCC300 -210KE3 -PeriErr_Circuit2_Slave(16-31)A" : Word;
   //       "BW_ASi200 -MCC300 -210KE3 -PeriErr_Circuit2_Slave(0-15)B" : Word;
   //       "BW_ASi200 -MCC300 -210KE3 -PeriErr_Circuit2_Slave(16-31)B" : Word;
   //    END_STRUCT;
   //    "word" : Struct
   //       Line : Struct
   //          ProductionLine : Struct
   //             Conveyor : Array[_.gminProductionLine.._.gmaxProductionLine] of Word;
   //          END_STRUCT;
   //          EmptyLine : Struct
   //             Conveyor : Array[_.gminEmptyLine.._.gmaxEmptyLine] of Word;
   //          END_STRUCT;
   //          PackedLine : Struct
   //             Conveyor : Array[_.gminPackedLine.._.gmaxPackedLine] of Word;
   //          END_STRUCT;
   //       END_STRUCT;
   //    END_STRUCT;
   // END_VAR
BEGIN
END_DATA_BLOCK

DATA_BLOCK "IDB_ManualControl"   // DB50
// stored: InstanceOfName Global.FB_ManualControl, InstanceOfType FB, Namespace Global
"Global.FB_ManualControl"
   // VAR RETAIN
   //    "Counter" { S7_SetPoint := 'True'} : CTU_INT;
   // END_VAR
BEGIN
END_DATA_BLOCK

DATA_BLOCK "IDB_Flow_Test"   // DB46
// stored: InstanceOfName ProductionLine.Flow_Test, InstanceOfType FB, Namespace ProductionLine
"ProductionLine.Flow_Test"
   // VAR
   //    Start { S7_SetPoint := 'True'} : Bool;
   //    StartTest { S7_SetPoint := 'True'} : "ProductionLine.Test_Logic";
   //    GoToRightDP1 { S7_SetPoint := 'True'} : "ProductionLine.Test_Logic";
   //    ContinueStraightDP1 { S7_SetPoint := 'True'} : "ProductionLine.Test_Logic";
   //    ContinueStraightDP2 { S7_SetPoint := 'True'} : "ProductionLine.Test_Logic";
   //    GotorightDP2Thentoright { S7_SetPoint := 'True'} : "ProductionLine.Test_Logic";
   //    GotorightDP2ThentoLeft { S7_SetPoint := 'True'} : "ProductionLine.Test_Logic";
   //    ContinueStraightDP3 { S7_SetPoint := 'True'} : "ProductionLine.Test_Logic";
   //    ContinueStraightDP4 { S7_SetPoint := 'True'} : "ProductionLine.Test_Logic";
   //    GotoRightDP4 { S7_SetPoint := 'True'} : "ProductionLine.Test_Logic";
   //    "A1.13.1_Straight" { S7_SetPoint := 'True'} : "ProductionLine.Test_Logic";
   //    "A1.13.1_left" { S7_SetPoint := 'True'} : "ProductionLine.Test_Logic";
   //    R_TRIG_Instance { S7_SetPoint := 'True'} : R_TRIG;
   // END_VAR
BEGIN
END_DATA_BLOCK

DATA_BLOCK "IDB_FB_ToggleDir"   // DB47
// stored: InstanceOfName ProductionLine.FB_ToggleDir, InstanceOfType FB, Namespace ProductionLine
"ProductionLine.FB_ToggleDir"
   // VAR
   //    "A1.12.1" { S7_SetPoint := 'True'} : "Global.ToggelDir";
   //    CurrentExpedtionDirection : Struct
   //       Straight : Bool;
   //       Left : Bool;
   //       None : Bool;
   //    END_STRUCT;
   //    CurrentStraightTableselection : Struct
   //       Table1 : Bool;
   //       Table2 : Bool;
   //       Table3 : Bool;
   //       Table4 : Bool;
   //       Table5 : Bool;
   //       None : Bool;
   //    END_STRUCT;
   //    CurrentLeftTableselection : Struct
   //       Table1 : Bool;
   //       Table2 : Bool;
   //       Table3 : Bool;
   //       Table4 : Bool;
   //       Table5 : Bool;
   //       None : Bool;
   //    END_STRUCT;
   // END_VAR
BEGIN
END_DATA_BLOCK

DATA_BLOCK "IDB_BarcodeReader"   // DB29
// stored: InstanceOfName ProductionLine.BarcodeReader, InstanceOfType FB, Namespace ProductionLine
"ProductionLine.BarcodeReader"
   // VAR
   //    DP1 : "Global.DataMan262";
   //    DP2 : "Global.DataMan262";
   //    DP3 : "Global.DataMan262";
   //    DP4 : "Global.DataMan262";
   // END_VAR
BEGIN
END_DATA_BLOCK

DATA_BLOCK "IDB_FB_Technology"   // DB38
// stored: InstanceOfName ProductionLine.FB_Technology, InstanceOfType FB, Namespace ProductionLine
"ProductionLine.FB_Technology"
   // VAR
   //    IP11 : String;
   //    IP12 : String;
   //    IP21 : String;
   //    IP22 : String;
   //    IP23 : String;
   //    IP31 : String;
   //    IP32 : String;
   //    IP41 : String;
   //    IP42 : String;
   //    ComDownStream : Struct
   //       DP1 : Bool;
   //       DP2 : Bool;
   //       DP3 : Bool;
   //       DP4 : Bool;
   //    END_STRUCT;
   //    ComTimmerDP1 { S7_SetPoint := 'True'} : TON_TIME;
   //    ComTimmerDP2 { S7_SetPoint := 'True'} : TON_TIME;
   //    ComTimmerDP3 { S7_SetPoint := 'True'} : TON_TIME;
   //    ComTimmerDP4 { S7_SetPoint := 'True'} : TON_TIME;
   // END_VAR
BEGIN
END_DATA_BLOCK

DATA_BLOCK "IDB_OPC_Communication"   // DB42
// stored: InstanceOfName ProductionLine.FB_OPC_Communication, InstanceOfType FB, Namespace ProductionLine
"ProductionLine.FB_OPC_Communication"
   // VAR
   //    Communication_DP1 : "ProductionLine.FB_OPC_DestRequest";
   //    Communication_DP2 : "ProductionLine.FB_OPC_DestRequest";
   //    Communication_DP3 : "ProductionLine.FB_OPC_DestRequest";
   //    Communication_DP4 : "ProductionLine.FB_OPC_DestRequest";
   //    Communication_IP1 : "ProductionLine.FB_OPC_DestInfo";
   //    Communication_IP2 : "ProductionLine.FB_OPC_DestInfo";
   //    Communication_IP3 : "ProductionLine.FB_OPC_DestInfo";
   //    Communication_IP4 : "ProductionLine.FB_OPC_DestInfo";
   //    Communication_IP5 : "ProductionLine.FB_OPC_DestInfo";
   //    Communication_IP6 : "ProductionLine.FB_OPC_DestInfo";
   //    Communication_IP7 : "ProductionLine.FB_OPC_DestInfo";
   //    Communication_IP8 : "ProductionLine.FB_OPC_DestInfo";
   //    Communication_IP9 : "ProductionLine.FB_OPC_DestInfo";
   //    Communication_SYS_OP : "ProductionLine.FB_OPC_SysStatus";
   //    Communication_SYS_OP_Source { S7_SetPoint := 'True'} : "ProductionLine.OPC_SystemStatus";
   //    Communication_SYS_OP_Ack { S7_SetPoint := 'True'} : "ProductionLine.OPC_SystStatus_Ack";
   //    timPeriodicSend { S7_SetPoint := 'True'} : IEC_TIMER;
   //    timWatchdog { S7_SetPoint := 'True'} : IEC_TIMER;
   //    Communication_fault : Bool;
   // END_VAR
BEGIN
END_DATA_BLOCK

DATA_BLOCK "IDB_Segments_Status"   // DB45
// stored: InstanceOfName ProductionLine.FB_Segments, InstanceOfType FB, Namespace ProductionLine
"ProductionLine.FB_Segments"
   // VAR
   //    ConveyorID : Int;
   //    "Counter" : Int;
   //    FlowRackLoop1 : Array[_."B1.1.1".._."B1.23.1"] of Bool;
   //    FlowRackLoop2 : Array[_."B1.6.1".._."B1.18.1"] of Bool;
   //    Fragileloop1 : Array[_."D1.1.1".._."E1.6.1"] of Bool;
   //    Fragileloop2 : Array[_."D1.9.1".._."D1.10.1"] of Bool;
   //    cmp : Struct
   //       FlowRackLoop1 : Array[_."B1.1.1".._."B1.23.1"] of Bool;
   //       FlowRackLoop2 : Array[_."B1.6.1".._."B1.18.1"] of Bool;
   //       Fragileloop1 : Array[_."D1.1.1".._."E1.6.1"] of Bool;
   //       Fragileloop2 : Array[_."D1.9.1".._."D1.10.1"] of Bool;
   //    END_STRUCT;
   //    FlowRackLoopReadyToRun : Bool;
   //    FlowRackWorkPlaceLeftReadyToRun : Bool;
   //    FlowRackWorkPlaceRightReadyToRun : Bool;
   //    FragileloopReadyToRun : Bool;
   // END_VAR
BEGIN
END_DATA_BLOCK

DATA_BLOCK "IDB_ToteTracking"   // DB11
// stored: InstanceOfName ProductionLine.FB_ToteTracking, InstanceOfType FB, Namespace ProductionLine
"ProductionLine.FB_ToteTracking"
   // VAR
   //    ZoneBpJam_Occ : TON_TIME;
   //    ZoneBpJam_NotOcc { S7_SetPoint := 'True'} : TON_TIME;
   //    DivertToManual { S7_SetPoint := 'True'} : Bool;
   //    HoldDivertToManual : Bool;
   //    RT_Exit_1_ : Array[1..1] of R_TRIG;
   //    RT_Exit_2_ : Array[1..6] of R_TRIG;
   //    NoReadTote { S7_SetPoint := 'True'} : String;
   //    NoData : Array[1..6] of Bool;
   // END_VAR
BEGIN
END_DATA_BLOCK
